   ExchangeToChain.AlmOKImmStopChain := TRUE;
   MecDetector.ScOk := FALSE;
   MecDetector.CycleOn := FALSE;
   MecDetector.Work := FALSE;
   MecDetector.OkToStop := FALSE;
   MecDetector.AlmOk := TRUE;
   MecDetector.MouldClear := FALSE;
   MecDetector.OutChainObstruction := FALSE;
   MecDetector.Ons_TimeWork := FALSE;
   MecDetector.SingleCycle := FALSE;
   MecDetector.Input.EnaSel := FALSE;
   MecDetector.Input.OffMouNotOpeSid := FALSE;
   MecDetector.Input.OnMouNotOpeSid := FALSE;
   MecDetector.Input.Chk1NotOpeSid := FALSE;
   MecDetector.Input.Chk2NotOpeSid := FALSE;
   MecDetector.Input.OffMouOpeSid := FALSE;
   MecDetector.Input.OnMouOpeSid := FALSE;
   MecDetector.Input.Chk1OpeSid := FALSE;
   MecDetector.Input.Chk2OpeSid := FALSE;
   MecDetector.Output.EnaSelLgh := FALSE;
   MecDetector.Output.CmdOnMouNotOpeSid := FALSE;
   MecDetector.Output.CmdOnMouOpeSid := FALSE;
   MecDetector.Man.Ons_SingleCycle := FALSE;
   MecDetector.Man.CmdSingleCycle := FALSE;
   MecDetector.Man.CmdOnMou := FALSE;
   MecDetector.Man.CmdOffMou := FALSE;
   MecDetector.Man.EnaPbt := FALSE;
   MecDetector.Man.RstCmd := FALSE;
   MecDetector.Man.ScreenNumber := 302_010_301;
   MecDetector.Man.WithinScreenRange := 0;
   MecDetector."Step"._00_CycleActivated_OnMouCmd := FALSE;
   MecDetector."Step"._10_OnMouPos_CheckResult := FALSE;
   MecDetector."Step"._20_ResultDone_OffMouCmd := FALSE;
   MecDetector."Step"._30_OffMouPos_EndCycle := FALSE;
   MecDetector."Step".Ons_StrobeWorkDone := FALSE;
   MecDetector."Step".StrobeWorkDone := FALSE;
   MecDetector."Step".ScSeqOk := FALSE;
   MecDetector."Step".SeqActive := FALSE;
   MecDetector."Step".TON_CheckResult.PT := T#500MS;
   MecDetector."Step".TON_CheckResult.IN := FALSE;
   MecDetector.RTO_Work.PT := T#1M;
   MecDetector.RTO_Work.IN := FALSE;
   MecDetector.TON_ScOK.PT := T#20S;
   MecDetector.TON_ScOK.IN := FALSE;
   MecDetector.TON_TimeoutWork.PT := T#20S;
   MecDetector.TON_TimeoutWork.IN := FALSE;
   MecDetector.TON_IncorrectPosOpeSide.PT := T#5S;
   MecDetector.TON_IncorrectPosOpeSide.IN := FALSE;
   MecDetector.TON_IncorrectPosNotOpeSide.PT := T#5S;
   MecDetector.TON_IncorrectPosNotOpeSide.IN := FALSE;
   MecDetector.TON_IncorrectPosPlate.PT := T#2S;
   MecDetector.TON_IncorrectPosPlate.IN := FALSE;
   OptDetector.ScOk := TRUE;
   OptDetector.CycleOn := FALSE;
   OptDetector.Work := FALSE;
   OptDetector.OkToStop := TRUE;
   OptDetector.AlmOk := TRUE;
   OptDetector.OutChainObstruction := TRUE;
   OptDetector.Ons_TimeWork := TRUE;
   OptDetector.Ons_ConnectionOn := FALSE;
   OptDetector.Ons_ChangeFormat := FALSE;
   OptDetector.Ons_RetrieveFormat := FALSE;
   OptDetector.RejectByDetector := FALSE;
   OptDetector.SingleCycle := FALSE;
   OptDetector.Ready := FALSE;
   OptDetector.SceneOk := FALSE;
   OptDetector.ChangeScene := FALSE;
   OptDetector.PhotoRequest := FALSE;
   OptDetector.SceneNumber := 0;
   OptDetector.Input.EnaSel := FALSE;
   OptDetector.Input.BrkSrs := TRUE;
   OptDetector.Input.Rdy := FALSE;
   OptDetector.Input.Brk := TRUE;
   OptDetector.Input.Run := TRUE;
   OptDetector.Input.Bsy := FALSE;
   OptDetector.Input.MouOk := FALSE;
   OptDetector.Input.Flt := FALSE;
   OptDetector.Input.WrkDone := FALSE;
   OptDetector.Input.FbkScn := 3;
   OptDetector.Output.EnaSelLgh := FALSE;
   OptDetector.Output.Lgh := FALSE;
   OptDetector.Output.CmdScnBit0 := TRUE;
   OptDetector.Output.CmdScnBit1 := FALSE;
   OptDetector.Output.CmdChgScn := FALSE;
   OptDetector.Output.CmdWrk := FALSE;
   OptDetector.Output.CmdRbo := FALSE;
   OptDetector.Output.CmdScn := 0;
   OptDetector.Man.Ons_SingleCycle := FALSE;
   OptDetector.Man.CmdSingleCycle := FALSE;
   OptDetector.Man.CmdStrobePhoto := FALSE;
   OptDetector.Man.EnaPbt := FALSE;
   OptDetector.Man.RstCmd := TRUE;
   OptDetector.Man.ScreenNumber := 302_020_301;
   OptDetector.Man.WithinScreenRange := 0;
   OptDetector."Step"._00_CycleActivated_StrobePhotoCmd := FALSE;
   OptDetector."Step"._10_ResultReady := FALSE;
   OptDetector."Step"._20_EndCycle := FALSE;
   OptDetector."Step".ons_StrobeWorkDone := FALSE;
   OptDetector."Step".StrobeWorkDone := FALSE;
   OptDetector."Step".ScSeqOk := FALSE;
   OptDetector."Step".SeqActive := FALSE;
   OptDetector.RTO_Work.PT := T#1M;
   OptDetector.RTO_Work.IN := FALSE;
   OptDetector.TON_ScOK.PT := T#20S;
   OptDetector.TON_ScOK.IN := FALSE;
   OptDetector.TON_TimeoutWork.PT := T#20S;
   OptDetector.TON_TimeoutWork.IN := FALSE;
   OptDetector.TON_TimeoutBusy.PT := T#5S;
   OptDetector.TON_TimeoutBusy.IN := FALSE;
   OptDetector.TON_TimeoutFormat.PT := T#5S;
   OptDetector.TON_TimeoutFormat.IN := FALSE;
   OptDetector.TOF_Ready.PT := T#500MS;
   OptDetector.TOF_Ready.ET := T#500MS;
   OptDetector.TOF_Ready.IN := FALSE;
   PusherExtractor.ScOk := FALSE;
   PusherExtractor.CycleOn := FALSE;
   PusherExtractor.Work := FALSE;
   PusherExtractor.OkToStop := FALSE;
   PusherExtractor.AlmOk := TRUE;
   PusherExtractor.DrivesEnabled := FALSE;
   PusherExtractor.OutChainObstruction := FALSE;
   PusherExtractor.SingleCycle := FALSE;
   PusherExtractor.RepositioningReq := FALSE;
   PusherExtractor.Ons_TimeWork := FALSE;
   PusherExtractor.NumMaxLevel := 0;
   PusherExtractor.Input.EnaSel := FALSE;
   PusherExtractor.Input.MaxLvl := FALSE;
   PusherExtractor.Input.HldOpnNotOpeSid := FALSE;
   PusherExtractor.Input.HldClsNotOpeSid := FALSE;
   PusherExtractor.Input.HldOpnOpeSid := FALSE;
   PusherExtractor.Input.HldClsOpeSid := FALSE;
   PusherExtractor.Output.EnaSelLgh := FALSE;
   PusherExtractor.Output.HldOpnNotOpeSid := FALSE;
   PusherExtractor.Output.HldClsNotOpeSid := FALSE;
   PusherExtractor.Output.HldOpnOpeSid := FALSE;
   PusherExtractor.Output.HldClsOpeSid := FALSE;
   PusherExtractor.Man.Ons_SingleCycle := FALSE;
   PusherExtractor.Man.CmdSupportOpen := FALSE;
   PusherExtractor.Man.CmdSupportClose := FALSE;
   PusherExtractor.Man.CmdSingleCycle := FALSE;
   PusherExtractor.Man.EnaPbt := FALSE;
   PusherExtractor.Man.RstCmd := FALSE;
   PusherExtractor.Man.ScreenNumber := 302_030_301;
   PusherExtractor.Man.WithinScreenRange := 0;
   PusherExtractor."Step"._00_CycleActived_UpCmd := FALSE;
   PusherExtractor."Step"._10_UpPos_IntermediateCmd := FALSE;
   PusherExtractor."Step"._20_IntermediatePos_OpenSupportCmd := FALSE;
   PusherExtractor."Step"._30_OpenSupportPos_DownCmd := FALSE;
   PusherExtractor."Step"._40_DownPos_CloseSupportCmd := FALSE;
   PusherExtractor."Step"._50_CloseSupportPos_CycleEnd := FALSE;
   PusherExtractor."Step".Ons_StrobeWorkDone := FALSE;
   PusherExtractor."Step".StrobeWorkDone := FALSE;
   PusherExtractor."Step".ScSeqOk := FALSE;
   PusherExtractor."Step".SeqActive := FALSE;
   PusherExtractor.Drive.AlmOk := FALSE;
   PusherExtractor.Drive.AlmEmerg := FALSE;
   PusherExtractor.Drive.AlmNode := FALSE;
   PusherExtractor.Drive.InitPosDrive := FALSE;
   PusherExtractor.Drive.InitPosDrivePLS := FALSE;
   PusherExtractor.Drive.GearingON := FALSE;
   PusherExtractor.Drive.CamHook := FALSE;
   PusherExtractor.Drive.CamStoppingPhase := FALSE;
   PusherExtractor.Drive.RepositioningRequest := FALSE;
   PusherExtractor.Drive.CamRequestResult := FALSE;
   PusherExtractor.Drive.CamRequestError := FALSE;
   PusherExtractor.Drive.CamRequestOk := FALSE;
   PusherExtractor.Drive.CalibDisAxisReq := FALSE;
   PusherExtractor.Drive.CalibReq := FALSE;
   PusherExtractor.Drive.CalibProcess := FALSE;
   PusherExtractor.Drive.HwOvertravelDisReq := FALSE;
   PusherExtractor.Drive.HwOvertravelEnReq := FALSE;
   PusherExtractor.Drive.AuxCamRequest := FALSE;
   PusherExtractor.Drive.TorquePeakEna := FALSE;
   PusherExtractor.Drive.Cmd_Repos := FALSE;
   PusherExtractor.Drive.Ons_CamRequest := FALSE;
   PusherExtractor.Drive.AuxCmdPosition := 0;
   PusherExtractor.Drive.Unwind := 0.0;
   PusherExtractor.Drive.MaxDev := 0.0;
   PusherExtractor.Drive.ReposSpeed := 100.0;
   PusherExtractor.Drive.CalcSlaveDifferenceABS := 0.0;
   PusherExtractor.Drive.CalcModPosition := 0.0;
   PusherExtractor.Drive.CalcSlaveDifference := 0.0;
   PusherExtractor.Drive.CalcMinDeltaPos := 0.0;
   PusherExtractor.Drive.CalcMaxDeltaPos := 0.0;
   PusherExtractor.Drive.CalcHalfPosUnwind := 0.0;
   PusherExtractor.Drive.Man.Cmd_PosJog := FALSE;
   PusherExtractor.Drive.Man.Cmd_NegJog := FALSE;
   PusherExtractor.Drive.Man.Cmd_Step := FALSE;
   PusherExtractor.Drive.Man.Cmd_Forward := FALSE;
   PusherExtractor.Drive.Man.Cmd_Backward := FALSE;
   PusherExtractor.Drive.Man.Cmd_Up := FALSE;
   PusherExtractor.Drive.Man.Cmd_Down := FALSE;
   PusherExtractor.Drive.Man.Cmd_Intermediate := FALSE;
   PusherExtractor.Drive.Man.Cmd_Open := FALSE;
   PusherExtractor.Drive.Man.Cmd_Close := FALSE;
   PusherExtractor.Drive.Man.Cmd_PreOpen := FALSE;
   PusherExtractor.Drive.Man.Cmd_Maintenance := FALSE;
   PusherExtractor.Drive.Man.Cmd_OperatorSide := FALSE;
   PusherExtractor.Drive.Man.Cmd_NotOperatorSide := FALSE;
   PusherExtractor.Drive.Man.Cmd_OnMould := FALSE;
   PusherExtractor.Drive.Man.Cmd_OffMould := FALSE;
   PusherExtractor.Drive.Man.Cmd_Pos0 := FALSE;
   PusherExtractor.Drive.Man.Cmd_Pos1 := FALSE;
   PusherExtractor.Drive.Man.Cmd_Pos2 := FALSE;
   PusherExtractor.Drive.Man.Cmd_Pos3 := FALSE;
   PusherExtractor.Drive.Man.Cmd_Pos4 := FALSE;
   PusherExtractor.Drive.Man.Cmd_Pos5 := FALSE;
   PusherExtractor.Drive.Man.Ons_Step := FALSE;
   PusherExtractor.Drive.Man.PhaseJogCmd := FALSE;
   PusherExtractor.Drive.Man.CmdStartStep := FALSE;
   PusherExtractor.Drive.Man.CmdEndStep := FALSE;
   PusherExtractor.Drive.Man.StepCond := FALSE;
   PusherExtractor.Drive.Man.TON_DelayHomeCmd.PT := T#3S;
   PusherExtractor.Drive.Man.TON_DelayHomeCmd.IN := FALSE;
   PusherExtractor.Drive.Auto.Cmd_Step := FALSE;
   PusherExtractor.Drive.Auto.Cmd_StartStep := FALSE;
   PusherExtractor.Drive.Auto.Cmd_EndStep := FALSE;
   PusherExtractor.Drive.Auto.Cmd_Forward := FALSE;
   PusherExtractor.Drive.Auto.Cmd_Backward := FALSE;
   PusherExtractor.Drive.Auto.Cmd_Up := FALSE;
   PusherExtractor.Drive.Auto.Cmd_Down := FALSE;
   PusherExtractor.Drive.Auto.Cmd_Intermediate := FALSE;
   PusherExtractor.Drive.Auto.Cmd_Open := FALSE;
   PusherExtractor.Drive.Auto.Cmd_Close := FALSE;
   PusherExtractor.Drive.Auto.Cmd_PreOpen := FALSE;
   PusherExtractor.Drive.Auto.Cmd_Maintenance := FALSE;
   PusherExtractor.Drive.Auto.Cmd_OperatorSide := FALSE;
   PusherExtractor.Drive.Auto.Cmd_NotOperatorSide := FALSE;
   PusherExtractor.Drive.Auto.Cmd_OnMould := FALSE;
   PusherExtractor.Drive.Auto.Cmd_OffMould := FALSE;
   PusherExtractor.Drive.Auto.Cmd_Pos0 := FALSE;
   PusherExtractor.Drive.Auto.Cmd_Pos1 := FALSE;
   PusherExtractor.Drive.Auto.Cmd_Pos2 := FALSE;
   PusherExtractor.Drive.Auto.Cmd_Pos3 := FALSE;
   PusherExtractor.Drive.Auto.Cmd_Pos4 := FALSE;
   PusherExtractor.Drive.Auto.Cmd_Pos5 := FALSE;
   PusherExtractor.Drive.Auto.Cmd_Gear := FALSE;
   PusherExtractor.Drive.ACT.CMD.Enable := FALSE;
   PusherExtractor.Drive.ACT.CMD.Pos_Mode := FALSE;
   PusherExtractor.Drive.ACT.CMD.MergeDisabled := FALSE;
   PusherExtractor.Drive.ACT.CMD.SCurve := FALSE;
   PusherExtractor.Drive.ACT.CMD.Cam_Mode := FALSE;
   PusherExtractor.Drive.ACT.CMD.Cam_Request := FALSE;
   PusherExtractor.Drive.ACT.CMD.Cam_PhaseStop := FALSE;
   PusherExtractor.Drive.ACT.CMD.Gear_Mode := FALSE;
   PusherExtractor.Drive.ACT.CMD.Repos_Req := FALSE;
   PusherExtractor.Drive.ACT.CMD.Jog_Pos := FALSE;
   PusherExtractor.Drive.ACT.CMD.Jog_Neg := FALSE;
   PusherExtractor.Drive.ACT.CMD.Stop := FALSE;
   PusherExtractor.Drive.ACT.CMD.Calibration_Req := FALSE;
   PusherExtractor.Drive.ACT.CMD.Reset := FALSE;
   PusherExtractor.Drive.ACT.CMD.RegInput1 := FALSE;
   PusherExtractor.Drive.ACT.CMD.Brake_Release := FALSE;
   PusherExtractor.Drive.ACT.CMD.HwPosOvertravel_Dis := FALSE;
   PusherExtractor.Drive.ACT.CMD.HwNegOvertravel_Dis := FALSE;
   PusherExtractor.Drive.ACT.CMD.HwOvertravel_MSG_En := FALSE;
   PusherExtractor.Drive.ACT.CMD.OneShootMove := FALSE;
   PusherExtractor.Drive.ACT.CMD.Move_Type := 0;
   PusherExtractor.Drive.ACT.CMD.Target_Pos := 0.0;
   PusherExtractor.Drive.ACT.CMD.Speed := 0.0;
   PusherExtractor.Drive.ACT.CMD.Acceleration := 0.0;
   PusherExtractor.Drive.ACT.CMD.Deceleration := 0.0;
   PusherExtractor.Drive.ACT.CMD.Torque_Limit := 0.0;
   PusherExtractor.Drive.ACT.CMD.Gear_Ratio := 0.0;
   PusherExtractor.Drive.ACT.CMD.Mccp_Length := 0;
   PusherExtractor.Drive.ACT.CMD.Mccp_StartSlope := 0.0;
   PusherExtractor.Drive.ACT.CMD.Mccp_EndSlope := 0.0;
   PusherExtractor.Drive.ACT.CMD.Mapc_Direction := 0;
   PusherExtractor.Drive.ACT.CMD.Mapc_SlaveScaling := 0.0;
   PusherExtractor.Drive.ACT.CMD.Mapc_MasterScaling := 0.0;
   PusherExtractor.Drive.ACT.CMD.Mapc_MasterLockPosition := 0.0;
   PusherExtractor.Drive.ACT.CMD.Mapc_CamLockPosition := 0.0;
   PusherExtractor.Drive.ACT.CMD.Cam[0..39].leadingValueStart := 0.0;
   PusherExtractor.Drive.ACT.CMD.Cam[0..39].leadingValueEnd := 0.0;
   PusherExtractor.Drive.ACT.CMD.Cam[0..39].followingValueStart := 0.0;
   PusherExtractor.Drive.ACT.CMD.Cam[0..39].followingValueEnd := 0.0;
   PusherExtractor.Drive.ACT.CMD.Cam[0..39].geoVeloStart := 0.0;
   PusherExtractor.Drive.ACT.CMD.Cam[0..39].geoVeloEnd := 0.0;
   PusherExtractor.Drive.ACT.CMD.Cam[0..39].geoAccelStart := 0.0;
   PusherExtractor.Drive.ACT.CMD.Cam[0..39].geoAccelEnd := 0.0;
   PusherExtractor.Drive.ACT.CMD.Cam[0..39].geoJerkStart := 0.0;
   PusherExtractor.Drive.ACT.CMD.Cam[0..39].geoJerkEnd := 0.0;
   PusherExtractor.Drive.ACT.CMD.Cam[0..39].inflectionPointParameter := 0.5;
   PusherExtractor.Drive.ACT.CMD.Cam[0..39].modVeloTrapezoidParameter := 1.0;
   PusherExtractor.Drive.ACT.CMD.Cam[0..39].modSineMaxAccelCaStar := 0.0;
   PusherExtractor.Drive.ACT.CMD.Cam[0..39].camProfileType := 0;
   PusherExtractor.Drive.ACT.FBK.Ready := FALSE;
   PusherExtractor.Drive.ACT.FBK.Calibrated := FALSE;
   PusherExtractor.Drive.ACT.FBK.Fault := FALSE;
   PusherExtractor.Drive.ACT.FBK.ModuleConnFault := FALSE;
   PusherExtractor.Drive.ACT.FBK.In_Position := FALSE;
   PusherExtractor.Drive.ACT.FBK.Standstill := FALSE;
   PusherExtractor.Drive.ACT.FBK.Enabled := FALSE;
   PusherExtractor.Drive.ACT.FBK.BusReadyStatus := FALSE;
   PusherExtractor.Drive.ACT.FBK.BrakeReleased := FALSE;
   PusherExtractor.Drive.ACT.FBK.HwPosOvertravelDisabled := FALSE;
   PusherExtractor.Drive.ACT.FBK.HwNegOvertravelDisabled := FALSE;
   PusherExtractor.Drive.ACT.FBK.SafeOffStatus := FALSE;
   PusherExtractor.Drive.ACT.FBK.MaxTorqueLimit := FALSE;
   PusherExtractor.Drive.ACT.FBK.PosMerge_IP := FALSE;
   PusherExtractor.Drive.ACT.FBK.PosMerge_PC := FALSE;
   PusherExtractor.Drive.ACT.FBK.Gearing_IP := FALSE;
   PusherExtractor.Drive.ACT.FBK.Position := 0.0;
   PusherExtractor.Drive.ACT.FBK.Speed := 0.0;
   PusherExtractor.Drive.ACT.FBK.Torque := 0.0;
   PusherExtractor.Drive.ACT.FBK.RegInput1Pos := 0.0;
   PusherExtractor.Drive.ACT.FBK.SeqCamErrorCode := 0;
   PusherExtractor.Drive.ACT.FBK.SeqCamTargetPosMAM := 0.0;
   PusherExtractor.Drive.ACT.FBK.SeqCamStatus.EndSequence := FALSE;
   PusherExtractor.Drive.ACT.FBK.SeqCamStatus.EndSuccess := FALSE;
   PusherExtractor.Drive.ACT.FBK.SeqCamStatus.EndError := FALSE;
   PusherExtractor.Drive.ACT.FBK.SeqCamStatus.CamHook := FALSE;
   PusherExtractor.Drive.ACT.FBK.SeqCamStatus.BothMapc_IP := FALSE;
   PusherExtractor.Drive.ACT.FBK.SeqCamStatus.SlaveFwd := FALSE;
   PusherExtractor.Drive.ACT.FBK.SeqCamStatus.SlaveBwd := FALSE;
   PusherExtractor.Drive.ACT.FBK.SeqCamStatus.SlaveUnwind := FALSE;
   PusherExtractor.Drive.ACT.FBK.SeqCamStatus.WaitValidByOpe := FALSE;
   PusherExtractor.Drive.ACT.FBK.SeqCamStatus.MapcA_IP := FALSE;
   PusherExtractor.Drive.ACT.FBK.SeqCamStatus.MapcB_IP := FALSE;
   PusherExtractor.Drive.ACT.FBK.SeqCamStatus.MapcC_IP := FALSE;
   PusherExtractor.Drive.ACT.FBK.SeqCamStatus.CamOnce_PC := FALSE;
   PusherExtractor.Drive.ACT.FBK.SeqCamStatus.MaxDevError := FALSE;
   PusherExtractor.Drive.ACT.FBK.SeqCamStatus.PositionCamLockStatus := FALSE;
   PusherExtractor.Drive.ACT.FBK.SeqCamStatus.WaitRestart := FALSE;
   PusherExtractor.Drive.ACT.FBK.SeqCamStatus.Bit17 := FALSE;
   PusherExtractor.Drive.ACT.FBK.SeqCamStatus.Bit18 := FALSE;
   PusherExtractor.Drive.ACT.FBK.SeqCamStatus.Bit19 := FALSE;
   PusherExtractor.Drive.ACT.FBK.SeqCamStatus.Bit20 := FALSE;
   PusherExtractor.Drive.ACT.FBK.SeqCamStatus.Bit21 := FALSE;
   PusherExtractor.Drive.ACT.FBK.SeqCamStatus.Bit22 := FALSE;
   PusherExtractor.Drive.ACT.FBK.SeqCamStatus.Bit23 := FALSE;
   PusherExtractor.Drive.ACT.FBK.SeqCamStatus.Bit24 := FALSE;
   PusherExtractor.Drive.ACT.FBK.SeqCamStatus.Bit25 := FALSE;
   PusherExtractor.Drive.ACT.FBK.SeqCamStatus.Bit26 := FALSE;
   PusherExtractor.Drive.ACT.FBK.SeqCamStatus.Bit27 := FALSE;
   PusherExtractor.Drive.ACT.FBK.SeqCamStatus.Bit28 := FALSE;
   PusherExtractor.Drive.ACT.FBK.SeqCamStatus.Bit29 := FALSE;
   PusherExtractor.Drive.ACT.FBK.SeqCamStatus.Bit30 := FALSE;
   PusherExtractor.Drive.ACT.FBK.SeqCamStatus.Bit31 := FALSE;
   PusherExtractor.Drive.ACT.FBK.SeqCamStatus.Bit32 := FALSE;
   PusherExtractor.Drive.PLS.FinePosOk.LowLimit := 0.0;
   PusherExtractor.Drive.PLS.FinePosOk.HighLimit := 0.0;
   PusherExtractor.Drive.PLS.FinePosOk.Ok := FALSE;
   PusherExtractor.Drive.PLS.KeepPosOk.LowLimit := 0.0;
   PusherExtractor.Drive.PLS.KeepPosOk.HighLimit := 0.0;
   PusherExtractor.Drive.PLS.KeepPosOk.Ok := FALSE;
   PusherExtractor.Drive.PLS.Up.LowLimit := 0.0;
   PusherExtractor.Drive.PLS.Up.HighLimit := 0.0;
   PusherExtractor.Drive.PLS.Up.Ok := FALSE;
   PusherExtractor.Drive.PLS.Intermediate.LowLimit := 0.0;
   PusherExtractor.Drive.PLS.Intermediate.HighLimit := 0.0;
   PusherExtractor.Drive.PLS.Intermediate.Ok := FALSE;
   PusherExtractor.Drive.PLS.Down.LowLimit := 0.0;
   PusherExtractor.Drive.PLS.Down.HighLimit := 0.0;
   PusherExtractor.Drive.PLS.Down.Ok := FALSE;
   PusherExtractor.Drive.PLS.Forward.LowLimit := 0.0;
   PusherExtractor.Drive.PLS.Forward.HighLimit := 0.0;
   PusherExtractor.Drive.PLS.Forward.Ok := FALSE;
   PusherExtractor.Drive.PLS.Backward.LowLimit := 0.0;
   PusherExtractor.Drive.PLS.Backward.HighLimit := 0.0;
   PusherExtractor.Drive.PLS.Backward.Ok := FALSE;
   PusherExtractor.Drive.PLS.Open.LowLimit := 0.0;
   PusherExtractor.Drive.PLS.Open.HighLimit := 0.0;
   PusherExtractor.Drive.PLS.Open.Ok := FALSE;
   PusherExtractor.Drive.PLS.Close.LowLimit := 0.0;
   PusherExtractor.Drive.PLS.Close.HighLimit := 0.0;
   PusherExtractor.Drive.PLS.Close.Ok := FALSE;
   PusherExtractor.Drive.PLS.PreOpen.LowLimit := 0.0;
   PusherExtractor.Drive.PLS.PreOpen.HighLimit := 0.0;
   PusherExtractor.Drive.PLS.PreOpen.Ok := FALSE;
   PusherExtractor.Drive.PLS.Maintenance.LowLimit := 0.0;
   PusherExtractor.Drive.PLS.Maintenance.HighLimit := 0.0;
   PusherExtractor.Drive.PLS.Maintenance.Ok := FALSE;
   PusherExtractor.Drive.PLS.OperatorSide.LowLimit := 0.0;
   PusherExtractor.Drive.PLS.OperatorSide.HighLimit := 0.0;
   PusherExtractor.Drive.PLS.OperatorSide.Ok := FALSE;
   PusherExtractor.Drive.PLS.NotOperatorSide.LowLimit := 0.0;
   PusherExtractor.Drive.PLS.NotOperatorSide.HighLimit := 0.0;
   PusherExtractor.Drive.PLS.NotOperatorSide.Ok := FALSE;
   PusherExtractor.Drive.PLS.OnMould.LowLimit := 0.0;
   PusherExtractor.Drive.PLS.OnMould.HighLimit := 0.0;
   PusherExtractor.Drive.PLS.OnMould.Ok := FALSE;
   PusherExtractor.Drive.PLS.OffMould.LowLimit := 0.0;
   PusherExtractor.Drive.PLS.OffMould.HighLimit := 0.0;
   PusherExtractor.Drive.PLS.OffMould.Ok := FALSE;
   PusherExtractor.Drive.PLS.Pos0.LowLimit := 0.0;
   PusherExtractor.Drive.PLS.Pos0.HighLimit := 0.0;
   PusherExtractor.Drive.PLS.Pos0.Ok := FALSE;
   PusherExtractor.Drive.PLS.Pos1.LowLimit := 0.0;
   PusherExtractor.Drive.PLS.Pos1.HighLimit := 0.0;
   PusherExtractor.Drive.PLS.Pos1.Ok := FALSE;
   PusherExtractor.Drive.PLS.Pos2.LowLimit := 0.0;
   PusherExtractor.Drive.PLS.Pos2.HighLimit := 0.0;
   PusherExtractor.Drive.PLS.Pos2.Ok := FALSE;
   PusherExtractor.Drive.PLS.Pos3.LowLimit := 0.0;
   PusherExtractor.Drive.PLS.Pos3.HighLimit := 0.0;
   PusherExtractor.Drive.PLS.Pos3.Ok := FALSE;
   PusherExtractor.Drive.PLS.Pos4.LowLimit := 0.0;
   PusherExtractor.Drive.PLS.Pos4.HighLimit := 0.0;
   PusherExtractor.Drive.PLS.Pos4.Ok := FALSE;
   PusherExtractor.Drive.PLS.Pos5.LowLimit := 0.0;
   PusherExtractor.Drive.PLS.Pos5.HighLimit := 0.0;
   PusherExtractor.Drive.PLS.Pos5.Ok := FALSE;
   PusherExtractor.Drive.TON_EnableDrive.PT := T#500MS;
   PusherExtractor.Drive.TON_EnableDrive.IN := FALSE;
   PusherExtractor.Drive.TON_HwOvertravel_Dis.PT := T#0MS;
   PusherExtractor.Drive.TON_HwOvertravel_Dis.IN := FALSE;
   PusherExtractor.Drive.TON_HwOvertravel_En.PT := T#0MS;
   PusherExtractor.Drive.TON_HwOvertravel_En.IN := FALSE;
   PusherExtractor.Drive.TON_TimeoutMovement.PT := T#8S;
   PusherExtractor.Drive.TON_TimeoutMovement.IN := FALSE;
   PusherExtractor.TON_ResetMaxLevel.PT := T#2S;
   PusherExtractor.TON_ResetMaxLevel.IN := FALSE;
   PusherExtractor.RTO_Work.PT := T#1M;
   PusherExtractor.RTO_Work.IN := FALSE;
   PusherExtractor.TON_ScOK.PT := T#20S;
   PusherExtractor.TON_ScOK.IN := FALSE;
   PusherExtractor.TON_IncorrectPosOpeSide.PT := T#4S;
   PusherExtractor.TON_IncorrectPosOpeSide.IN := FALSE;
   PusherExtractor.TON_IncorrectPosNotOpeSide.PT := T#4S;
   PusherExtractor.TON_IncorrectPosNotOpeSide.IN := FALSE;
   PusherExtractor.TON_Sign_MaxLevel.PT := T#1S;
   PusherExtractor.TON_Sign_MaxLevel.IN := FALSE;
   PusherExtractor.TON_TimeoutWork.PT := T#20S;
   PusherExtractor.TON_TimeoutWork.IN := FALSE;
   RotaryExtractor.ScOk := FALSE;
   RotaryExtractor.CycleOn := FALSE;
   RotaryExtractor.Work := FALSE;
   RotaryExtractor.OkToStop := TRUE;
   RotaryExtractor.AlmOk := TRUE;
   RotaryExtractor.DrivesEnabled := FALSE;
   RotaryExtractor.OutChainObstruction := TRUE;
   RotaryExtractor.RepositioningReq := FALSE;
   RotaryExtractor.Ons_TimeWork := TRUE;
   RotaryExtractor.NumMaxLevel := 0;
   RotaryExtractor.Input.EnaSel := FALSE;
   RotaryExtractor.Input.MaxLvl := FALSE;
   RotaryExtractor.Output.EnaSelLgh := FALSE;
   RotaryExtractor.Man.EnaPbt := FALSE;
   RotaryExtractor.Man.RstCmd := TRUE;
   RotaryExtractor.Man.ScreenNumber := 302_040_301;
   RotaryExtractor.Man.WithinScreenRange := 0;
   RotaryExtractor."Step"._00_CycleActived_StartRotationCmd := FALSE;
   RotaryExtractor."Step"._10_RotationOutPos_StopRotationCmd := FALSE;
   RotaryExtractor."Step"._20_FinePos_CycleEnd := FALSE;
   RotaryExtractor."Step".Ons_StrobeWorkDone := FALSE;
   RotaryExtractor."Step".StrobeWorkDone := FALSE;
   RotaryExtractor."Step".ScSeqOk := FALSE;
   RotaryExtractor."Step".SeqActive := FALSE;
   RotaryExtractor.Drive.AlmOk := FALSE;
   RotaryExtractor.Drive.AlmEmerg := FALSE;
   RotaryExtractor.Drive.AlmNode := FALSE;
   RotaryExtractor.Drive.InitPosDrive := FALSE;
   RotaryExtractor.Drive.InitPosDrivePLS := FALSE;
   RotaryExtractor.Drive.GearingON := FALSE;
   RotaryExtractor.Drive.CamHook := FALSE;
   RotaryExtractor.Drive.CamStoppingPhase := FALSE;
   RotaryExtractor.Drive.RepositioningRequest := FALSE;
   RotaryExtractor.Drive.CamRequestResult := FALSE;
   RotaryExtractor.Drive.CamRequestError := FALSE;
   RotaryExtractor.Drive.CamRequestOk := FALSE;
   RotaryExtractor.Drive.CalibDisAxisReq := FALSE;
   RotaryExtractor.Drive.CalibReq := FALSE;
   RotaryExtractor.Drive.CalibProcess := FALSE;
   RotaryExtractor.Drive.HwOvertravelDisReq := FALSE;
   RotaryExtractor.Drive.HwOvertravelEnReq := FALSE;
   RotaryExtractor.Drive.AuxCamRequest := FALSE;
   RotaryExtractor.Drive.TorquePeakEna := TRUE;
   RotaryExtractor.Drive.Cmd_Repos := FALSE;
   RotaryExtractor.Drive.Ons_CamRequest := FALSE;
   RotaryExtractor.Drive.AuxCmdPosition := 0;
   RotaryExtractor.Drive.Unwind := 120.0;
   RotaryExtractor.Drive.MaxDev := 0.0;
   RotaryExtractor.Drive.ReposSpeed := 100.0;
   RotaryExtractor.Drive.CalcSlaveDifferenceABS := 0.0;
   RotaryExtractor.Drive.CalcModPosition := 0.0;
   RotaryExtractor.Drive.CalcSlaveDifference := 0.0;
   RotaryExtractor.Drive.CalcMinDeltaPos := 0.0;
   RotaryExtractor.Drive.CalcMaxDeltaPos := 0.0;
   RotaryExtractor.Drive.CalcHalfPosUnwind := 0.0;
   RotaryExtractor.Drive.Man.Cmd_PosJog := FALSE;
   RotaryExtractor.Drive.Man.Cmd_NegJog := FALSE;
   RotaryExtractor.Drive.Man.Cmd_Step := FALSE;
   RotaryExtractor.Drive.Man.Cmd_Forward := FALSE;
   RotaryExtractor.Drive.Man.Cmd_Backward := FALSE;
   RotaryExtractor.Drive.Man.Cmd_Up := FALSE;
   RotaryExtractor.Drive.Man.Cmd_Down := FALSE;
   RotaryExtractor.Drive.Man.Cmd_Intermediate := FALSE;
   RotaryExtractor.Drive.Man.Cmd_Open := FALSE;
   RotaryExtractor.Drive.Man.Cmd_Close := FALSE;
   RotaryExtractor.Drive.Man.Cmd_PreOpen := FALSE;
   RotaryExtractor.Drive.Man.Cmd_Maintenance := FALSE;
   RotaryExtractor.Drive.Man.Cmd_OperatorSide := FALSE;
   RotaryExtractor.Drive.Man.Cmd_NotOperatorSide := FALSE;
   RotaryExtractor.Drive.Man.Cmd_OnMould := FALSE;
   RotaryExtractor.Drive.Man.Cmd_OffMould := FALSE;
   RotaryExtractor.Drive.Man.Cmd_Pos0 := FALSE;
   RotaryExtractor.Drive.Man.Cmd_Pos1 := FALSE;
   RotaryExtractor.Drive.Man.Cmd_Pos2 := FALSE;
   RotaryExtractor.Drive.Man.Cmd_Pos3 := FALSE;
   RotaryExtractor.Drive.Man.Cmd_Pos4 := FALSE;
   RotaryExtractor.Drive.Man.Cmd_Pos5 := FALSE;
   RotaryExtractor.Drive.Man.Ons_Step := FALSE;
   RotaryExtractor.Drive.Man.PhaseJogCmd := FALSE;
   RotaryExtractor.Drive.Man.CmdStartStep := FALSE;
   RotaryExtractor.Drive.Man.CmdEndStep := FALSE;
   RotaryExtractor.Drive.Man.StepCond := FALSE;
   RotaryExtractor.Drive.Man.TON_DelayHomeCmd.PT := T#3S;
   RotaryExtractor.Drive.Man.TON_DelayHomeCmd.IN := FALSE;
   RotaryExtractor.Drive.Auto.Cmd_Step := FALSE;
   RotaryExtractor.Drive.Auto.Cmd_StartStep := FALSE;
   RotaryExtractor.Drive.Auto.Cmd_EndStep := FALSE;
   RotaryExtractor.Drive.Auto.Cmd_Forward := FALSE;
   RotaryExtractor.Drive.Auto.Cmd_Backward := FALSE;
   RotaryExtractor.Drive.Auto.Cmd_Up := FALSE;
   RotaryExtractor.Drive.Auto.Cmd_Down := FALSE;
   RotaryExtractor.Drive.Auto.Cmd_Intermediate := FALSE;
   RotaryExtractor.Drive.Auto.Cmd_Open := FALSE;
   RotaryExtractor.Drive.Auto.Cmd_Close := FALSE;
   RotaryExtractor.Drive.Auto.Cmd_PreOpen := FALSE;
   RotaryExtractor.Drive.Auto.Cmd_Maintenance := FALSE;
   RotaryExtractor.Drive.Auto.Cmd_OperatorSide := FALSE;
   RotaryExtractor.Drive.Auto.Cmd_NotOperatorSide := FALSE;
   RotaryExtractor.Drive.Auto.Cmd_OnMould := FALSE;
   RotaryExtractor.Drive.Auto.Cmd_OffMould := FALSE;
   RotaryExtractor.Drive.Auto.Cmd_Pos0 := FALSE;
   RotaryExtractor.Drive.Auto.Cmd_Pos1 := FALSE;
   RotaryExtractor.Drive.Auto.Cmd_Pos2 := FALSE;
   RotaryExtractor.Drive.Auto.Cmd_Pos3 := FALSE;
   RotaryExtractor.Drive.Auto.Cmd_Pos4 := FALSE;
   RotaryExtractor.Drive.Auto.Cmd_Pos5 := FALSE;
   RotaryExtractor.Drive.Auto.Cmd_Gear := FALSE;
   RotaryExtractor.Drive.ACT.CMD.Enable := FALSE;
   RotaryExtractor.Drive.ACT.CMD.Pos_Mode := FALSE;
   RotaryExtractor.Drive.ACT.CMD.MergeDisabled := FALSE;
   RotaryExtractor.Drive.ACT.CMD.SCurve := FALSE;
   RotaryExtractor.Drive.ACT.CMD.Cam_Mode := FALSE;
   RotaryExtractor.Drive.ACT.CMD.Cam_Request := FALSE;
   RotaryExtractor.Drive.ACT.CMD.Cam_PhaseStop := FALSE;
   RotaryExtractor.Drive.ACT.CMD.Gear_Mode := FALSE;
   RotaryExtractor.Drive.ACT.CMD.Repos_Req := FALSE;
   RotaryExtractor.Drive.ACT.CMD.Jog_Pos := FALSE;
   RotaryExtractor.Drive.ACT.CMD.Jog_Neg := FALSE;
   RotaryExtractor.Drive.ACT.CMD.Stop := TRUE;
   RotaryExtractor.Drive.ACT.CMD.Calibration_Req := FALSE;
   RotaryExtractor.Drive.ACT.CMD.Reset := FALSE;
   RotaryExtractor.Drive.ACT.CMD.RegInput1 := FALSE;
   RotaryExtractor.Drive.ACT.CMD.Brake_Release := FALSE;
   RotaryExtractor.Drive.ACT.CMD.HwPosOvertravel_Dis := FALSE;
   RotaryExtractor.Drive.ACT.CMD.HwNegOvertravel_Dis := FALSE;
   RotaryExtractor.Drive.ACT.CMD.HwOvertravel_MSG_En := FALSE;
   RotaryExtractor.Drive.ACT.CMD.OneShootMove := FALSE;
   RotaryExtractor.Drive.ACT.CMD.Move_Type := 0;
   RotaryExtractor.Drive.ACT.CMD.Target_Pos := 0.0;
   RotaryExtractor.Drive.ACT.CMD.Speed := 0.0;
   RotaryExtractor.Drive.ACT.CMD.Acceleration := 0.0;
   RotaryExtractor.Drive.ACT.CMD.Deceleration := 4500.0;
   RotaryExtractor.Drive.ACT.CMD.Torque_Limit := 30.0;
   RotaryExtractor.Drive.ACT.CMD.Gear_Ratio := 0.0;
   RotaryExtractor.Drive.ACT.CMD.Mccp_Length := 0;
   RotaryExtractor.Drive.ACT.CMD.Mccp_StartSlope := 0.0;
   RotaryExtractor.Drive.ACT.CMD.Mccp_EndSlope := 0.0;
   RotaryExtractor.Drive.ACT.CMD.Mapc_Direction := 0;
   RotaryExtractor.Drive.ACT.CMD.Mapc_SlaveScaling := 0.0;
   RotaryExtractor.Drive.ACT.CMD.Mapc_MasterScaling := 0.0;
   RotaryExtractor.Drive.ACT.CMD.Mapc_MasterLockPosition := 0.0;
   RotaryExtractor.Drive.ACT.CMD.Mapc_CamLockPosition := 0.0;
   RotaryExtractor.Drive.ACT.CMD.Cam[0..39].leadingValueStart := 0.0;
   RotaryExtractor.Drive.ACT.CMD.Cam[0..39].leadingValueEnd := 0.0;
   RotaryExtractor.Drive.ACT.CMD.Cam[0..39].followingValueStart := 0.0;
   RotaryExtractor.Drive.ACT.CMD.Cam[0..39].followingValueEnd := 0.0;
   RotaryExtractor.Drive.ACT.CMD.Cam[0..39].geoVeloStart := 0.0;
   RotaryExtractor.Drive.ACT.CMD.Cam[0..39].geoVeloEnd := 0.0;
   RotaryExtractor.Drive.ACT.CMD.Cam[0..39].geoAccelStart := 0.0;
   RotaryExtractor.Drive.ACT.CMD.Cam[0..39].geoAccelEnd := 0.0;
   RotaryExtractor.Drive.ACT.CMD.Cam[0..39].geoJerkStart := 0.0;
   RotaryExtractor.Drive.ACT.CMD.Cam[0..39].geoJerkEnd := 0.0;
   RotaryExtractor.Drive.ACT.CMD.Cam[0..39].inflectionPointParameter := 0.5;
   RotaryExtractor.Drive.ACT.CMD.Cam[0..39].modVeloTrapezoidParameter := 1.0;
   RotaryExtractor.Drive.ACT.CMD.Cam[0..39].modSineMaxAccelCaStar := 0.0;
   RotaryExtractor.Drive.ACT.CMD.Cam[0..39].camProfileType := 0;
   RotaryExtractor.Drive.ACT.FBK.Ready := TRUE;
   RotaryExtractor.Drive.ACT.FBK.Calibrated := TRUE;
   RotaryExtractor.Drive.ACT.FBK.Fault := FALSE;
   RotaryExtractor.Drive.ACT.FBK.ModuleConnFault := FALSE;
   RotaryExtractor.Drive.ACT.FBK.In_Position := FALSE;
   RotaryExtractor.Drive.ACT.FBK.Standstill := TRUE;
   RotaryExtractor.Drive.ACT.FBK.Enabled := FALSE;
   RotaryExtractor.Drive.ACT.FBK.BusReadyStatus := FALSE;
   RotaryExtractor.Drive.ACT.FBK.BrakeReleased := FALSE;
   RotaryExtractor.Drive.ACT.FBK.HwPosOvertravelDisabled := FALSE;
   RotaryExtractor.Drive.ACT.FBK.HwNegOvertravelDisabled := FALSE;
   RotaryExtractor.Drive.ACT.FBK.SafeOffStatus := FALSE;
   RotaryExtractor.Drive.ACT.FBK.MaxTorqueLimit := FALSE;
   RotaryExtractor.Drive.ACT.FBK.PosMerge_IP := FALSE;
   RotaryExtractor.Drive.ACT.FBK.PosMerge_PC := FALSE;
   RotaryExtractor.Drive.ACT.FBK.Gearing_IP := FALSE;
   RotaryExtractor.Drive.ACT.FBK.Position := 0.003;
   RotaryExtractor.Drive.ACT.FBK.Speed := 0.0;
   RotaryExtractor.Drive.ACT.FBK.Torque := 0.0;
   RotaryExtractor.Drive.ACT.FBK.RegInput1Pos := 0.0;
   RotaryExtractor.Drive.ACT.FBK.SeqCamErrorCode := 0;
   RotaryExtractor.Drive.ACT.FBK.SeqCamTargetPosMAM := 0.0;
   RotaryExtractor.Drive.ACT.FBK.SeqCamStatus.EndSequence := FALSE;
   RotaryExtractor.Drive.ACT.FBK.SeqCamStatus.EndSuccess := FALSE;
   RotaryExtractor.Drive.ACT.FBK.SeqCamStatus.EndError := FALSE;
   RotaryExtractor.Drive.ACT.FBK.SeqCamStatus.CamHook := FALSE;
   RotaryExtractor.Drive.ACT.FBK.SeqCamStatus.BothMapc_IP := FALSE;
   RotaryExtractor.Drive.ACT.FBK.SeqCamStatus.SlaveFwd := FALSE;
   RotaryExtractor.Drive.ACT.FBK.SeqCamStatus.SlaveBwd := FALSE;
   RotaryExtractor.Drive.ACT.FBK.SeqCamStatus.SlaveUnwind := FALSE;
   RotaryExtractor.Drive.ACT.FBK.SeqCamStatus.WaitValidByOpe := FALSE;
   RotaryExtractor.Drive.ACT.FBK.SeqCamStatus.MapcA_IP := FALSE;
   RotaryExtractor.Drive.ACT.FBK.SeqCamStatus.MapcB_IP := FALSE;
   RotaryExtractor.Drive.ACT.FBK.SeqCamStatus.MapcC_IP := FALSE;
   RotaryExtractor.Drive.ACT.FBK.SeqCamStatus.CamOnce_PC := FALSE;
   RotaryExtractor.Drive.ACT.FBK.SeqCamStatus.MaxDevError := FALSE;
   RotaryExtractor.Drive.ACT.FBK.SeqCamStatus.PositionCamLockStatus := FALSE;
   RotaryExtractor.Drive.ACT.FBK.SeqCamStatus.WaitRestart := FALSE;
   RotaryExtractor.Drive.ACT.FBK.SeqCamStatus.Bit17 := FALSE;
   RotaryExtractor.Drive.ACT.FBK.SeqCamStatus.Bit18 := FALSE;
   RotaryExtractor.Drive.ACT.FBK.SeqCamStatus.Bit19 := FALSE;
   RotaryExtractor.Drive.ACT.FBK.SeqCamStatus.Bit20 := FALSE;
   RotaryExtractor.Drive.ACT.FBK.SeqCamStatus.Bit21 := FALSE;
   RotaryExtractor.Drive.ACT.FBK.SeqCamStatus.Bit22 := FALSE;
   RotaryExtractor.Drive.ACT.FBK.SeqCamStatus.Bit23 := FALSE;
   RotaryExtractor.Drive.ACT.FBK.SeqCamStatus.Bit24 := FALSE;
   RotaryExtractor.Drive.ACT.FBK.SeqCamStatus.Bit25 := FALSE;
   RotaryExtractor.Drive.ACT.FBK.SeqCamStatus.Bit26 := FALSE;
   RotaryExtractor.Drive.ACT.FBK.SeqCamStatus.Bit27 := FALSE;
   RotaryExtractor.Drive.ACT.FBK.SeqCamStatus.Bit28 := FALSE;
   RotaryExtractor.Drive.ACT.FBK.SeqCamStatus.Bit29 := FALSE;
   RotaryExtractor.Drive.ACT.FBK.SeqCamStatus.Bit30 := FALSE;
   RotaryExtractor.Drive.ACT.FBK.SeqCamStatus.Bit31 := FALSE;
   RotaryExtractor.Drive.ACT.FBK.SeqCamStatus.Bit32 := FALSE;
   RotaryExtractor.Drive.PLS.FinePosOk.LowLimit := 119.0;
   RotaryExtractor.Drive.PLS.FinePosOk.HighLimit := 1.0;
   RotaryExtractor.Drive.PLS.FinePosOk.Ok := TRUE;
   RotaryExtractor.Drive.PLS.KeepPosOk.LowLimit := 0.0;
   RotaryExtractor.Drive.PLS.KeepPosOk.HighLimit := 0.0;
   RotaryExtractor.Drive.PLS.KeepPosOk.Ok := FALSE;
   RotaryExtractor.Drive.PLS.Up.LowLimit := 0.0;
   RotaryExtractor.Drive.PLS.Up.HighLimit := 0.0;
   RotaryExtractor.Drive.PLS.Up.Ok := FALSE;
   RotaryExtractor.Drive.PLS.Intermediate.LowLimit := 0.0;
   RotaryExtractor.Drive.PLS.Intermediate.HighLimit := 0.0;
   RotaryExtractor.Drive.PLS.Intermediate.Ok := FALSE;
   RotaryExtractor.Drive.PLS.Down.LowLimit := 0.0;
   RotaryExtractor.Drive.PLS.Down.HighLimit := 0.0;
   RotaryExtractor.Drive.PLS.Down.Ok := FALSE;
   RotaryExtractor.Drive.PLS.Forward.LowLimit := 0.0;
   RotaryExtractor.Drive.PLS.Forward.HighLimit := 0.0;
   RotaryExtractor.Drive.PLS.Forward.Ok := FALSE;
   RotaryExtractor.Drive.PLS.Backward.LowLimit := 0.0;
   RotaryExtractor.Drive.PLS.Backward.HighLimit := 0.0;
   RotaryExtractor.Drive.PLS.Backward.Ok := FALSE;
   RotaryExtractor.Drive.PLS.Open.LowLimit := 0.0;
   RotaryExtractor.Drive.PLS.Open.HighLimit := 0.0;
   RotaryExtractor.Drive.PLS.Open.Ok := FALSE;
   RotaryExtractor.Drive.PLS.Close.LowLimit := 0.0;
   RotaryExtractor.Drive.PLS.Close.HighLimit := 0.0;
   RotaryExtractor.Drive.PLS.Close.Ok := FALSE;
   RotaryExtractor.Drive.PLS.PreOpen.LowLimit := 0.0;
   RotaryExtractor.Drive.PLS.PreOpen.HighLimit := 0.0;
   RotaryExtractor.Drive.PLS.PreOpen.Ok := FALSE;
   RotaryExtractor.Drive.PLS.Maintenance.LowLimit := 0.0;
   RotaryExtractor.Drive.PLS.Maintenance.HighLimit := 0.0;
   RotaryExtractor.Drive.PLS.Maintenance.Ok := FALSE;
   RotaryExtractor.Drive.PLS.OperatorSide.LowLimit := 0.0;
   RotaryExtractor.Drive.PLS.OperatorSide.HighLimit := 0.0;
   RotaryExtractor.Drive.PLS.OperatorSide.Ok := FALSE;
   RotaryExtractor.Drive.PLS.NotOperatorSide.LowLimit := 0.0;
   RotaryExtractor.Drive.PLS.NotOperatorSide.HighLimit := 0.0;
   RotaryExtractor.Drive.PLS.NotOperatorSide.Ok := FALSE;
   RotaryExtractor.Drive.PLS.OnMould.LowLimit := 0.0;
   RotaryExtractor.Drive.PLS.OnMould.HighLimit := 0.0;
   RotaryExtractor.Drive.PLS.OnMould.Ok := FALSE;
   RotaryExtractor.Drive.PLS.OffMould.LowLimit := 0.0;
   RotaryExtractor.Drive.PLS.OffMould.HighLimit := 0.0;
   RotaryExtractor.Drive.PLS.OffMould.Ok := FALSE;
   RotaryExtractor.Drive.PLS.Pos0.LowLimit := 60.0;
   RotaryExtractor.Drive.PLS.Pos0.HighLimit := 120.1;
   RotaryExtractor.Drive.PLS.Pos0.Ok := FALSE;
   RotaryExtractor.Drive.PLS.Pos1.LowLimit := 0.0;
   RotaryExtractor.Drive.PLS.Pos1.HighLimit := 0.0;
   RotaryExtractor.Drive.PLS.Pos1.Ok := FALSE;
   RotaryExtractor.Drive.PLS.Pos2.LowLimit := 0.0;
   RotaryExtractor.Drive.PLS.Pos2.HighLimit := 0.0;
   RotaryExtractor.Drive.PLS.Pos2.Ok := FALSE;
   RotaryExtractor.Drive.PLS.Pos3.LowLimit := 0.0;
   RotaryExtractor.Drive.PLS.Pos3.HighLimit := 0.0;
   RotaryExtractor.Drive.PLS.Pos3.Ok := FALSE;
   RotaryExtractor.Drive.PLS.Pos4.LowLimit := 0.0;
   RotaryExtractor.Drive.PLS.Pos4.HighLimit := 0.0;
   RotaryExtractor.Drive.PLS.Pos4.Ok := FALSE;
   RotaryExtractor.Drive.PLS.Pos5.LowLimit := 0.0;
   RotaryExtractor.Drive.PLS.Pos5.HighLimit := 0.0;
   RotaryExtractor.Drive.PLS.Pos5.Ok := FALSE;
   RotaryExtractor.Drive.TON_EnableDrive.PT := T#500MS;
   RotaryExtractor.Drive.TON_EnableDrive.IN := FALSE;
   RotaryExtractor.Drive.TON_HwOvertravel_Dis.PT := T#0MS;
   RotaryExtractor.Drive.TON_HwOvertravel_Dis.IN := FALSE;
   RotaryExtractor.Drive.TON_HwOvertravel_En.PT := T#0MS;
   RotaryExtractor.Drive.TON_HwOvertravel_En.IN := FALSE;
   RotaryExtractor.Drive.TON_TimeoutMovement.PT := T#8S;
   RotaryExtractor.Drive.TON_TimeoutMovement.IN := FALSE;
   RotaryExtractor.TON_ResetMaxLevel.PT := T#2S;
   RotaryExtractor.TON_ResetMaxLevel.ET := T#2S;
   RotaryExtractor.TON_ResetMaxLevel.IN := TRUE;
   RotaryExtractor.TON_ResetMaxLevel.Q := TRUE;
   RotaryExtractor.RTO_Work.PT := T#1M;
   RotaryExtractor.RTO_Work.IN := FALSE;
   RotaryExtractor.TON_ScOK.PT := T#20S;
   RotaryExtractor.TON_ScOK.IN := FALSE;
   RotaryExtractor.TON_Sign_MaxLevel.PT := T#1S;
   RotaryExtractor.TON_Sign_MaxLevel.IN := FALSE;
   RotaryExtractor.TON_TimeoutWork.PT := T#20S;
   RotaryExtractor.TON_TimeoutWork.IN := FALSE;
   PickExtractor.ScOk := FALSE;
   PickExtractor.CycleOn := FALSE;
   PickExtractor.Work := FALSE;
   PickExtractor.OkToStop := FALSE;
   PickExtractor.AlmOk := TRUE;
   PickExtractor.DrivesEnabled := FALSE;
   PickExtractor.OutChainObstruction := FALSE;
   PickExtractor.SingleCycle := FALSE;
   PickExtractor.RepositioningReq := FALSE;
   PickExtractor.Ons_TimeWork := FALSE;
   PickExtractor.NumMaxLevel := 0;
   PickExtractor.Input.EnaSel := FALSE;
   PickExtractor.Input.MaxLvl := FALSE;
   PickExtractor.Input.HldOpnNotOpeSid := FALSE;
   PickExtractor.Input.HldClsNotOpeSid := FALSE;
   PickExtractor.Input.HldOpnOpeSid := FALSE;
   PickExtractor.Input.HldClsOpeSid := FALSE;
   PickExtractor.Output.EnaSelLgh := FALSE;
   PickExtractor.Output.HldOpnNotOpeSid := FALSE;
   PickExtractor.Output.HldClsNotOpeSid := FALSE;
   PickExtractor.Output.HldOpnOpeSid := FALSE;
   PickExtractor.Output.HldClsOpeSid := FALSE;
   PickExtractor.Man.Ons_SingleCycle := FALSE;
   PickExtractor.Man.CmdSupportOpen := FALSE;
   PickExtractor.Man.CmdSupportClose := FALSE;
   PickExtractor.Man.CmdSingleCycle := FALSE;
   PickExtractor.Man.EnaPbt := FALSE;
   PickExtractor.Man.RstCmd := FALSE;
   PickExtractor.Man.ScreenNumber := 302_050_301;
   PickExtractor.Man.WithinScreenRange := 0;
   PickExtractor."Step"._00_CycleActived_IntermediateCmd := FALSE;
   PickExtractor."Step"._10_IntermediatePos_OpenSupportCmd := FALSE;
   PickExtractor."Step"._20_OpenSupportPos_DownCmd := FALSE;
   PickExtractor."Step"._30_DownPos_CloseSupportCmd := FALSE;
   PickExtractor."Step"._40_CloseSupportPos_CycleEnd := FALSE;
   PickExtractor."Step".Ons_StrobeWorkDone := FALSE;
   PickExtractor."Step".StrobeWorkDone := FALSE;
   PickExtractor."Step".ScSeqOk := FALSE;
   PickExtractor."Step".SeqActive := FALSE;
   PickExtractor.Drive.AlmOk := FALSE;
   PickExtractor.Drive.AlmEmerg := FALSE;
   PickExtractor.Drive.AlmNode := FALSE;
   PickExtractor.Drive.InitPosDrive := FALSE;
   PickExtractor.Drive.InitPosDrivePLS := FALSE;
   PickExtractor.Drive.GearingON := FALSE;
   PickExtractor.Drive.CamHook := FALSE;
   PickExtractor.Drive.CamStoppingPhase := FALSE;
   PickExtractor.Drive.RepositioningRequest := FALSE;
   PickExtractor.Drive.CamRequestResult := FALSE;
   PickExtractor.Drive.CamRequestError := FALSE;
   PickExtractor.Drive.CamRequestOk := FALSE;
   PickExtractor.Drive.CalibDisAxisReq := FALSE;
   PickExtractor.Drive.CalibReq := FALSE;
   PickExtractor.Drive.CalibProcess := FALSE;
   PickExtractor.Drive.HwOvertravelDisReq := FALSE;
   PickExtractor.Drive.HwOvertravelEnReq := FALSE;
   PickExtractor.Drive.AuxCamRequest := FALSE;
   PickExtractor.Drive.TorquePeakEna := FALSE;
   PickExtractor.Drive.Cmd_Repos := FALSE;
   PickExtractor.Drive.Ons_CamRequest := FALSE;
   PickExtractor.Drive.AuxCmdPosition := 0;
   PickExtractor.Drive.Unwind := 0.0;
   PickExtractor.Drive.MaxDev := 0.0;
   PickExtractor.Drive.ReposSpeed := 100.0;
   PickExtractor.Drive.CalcSlaveDifferenceABS := 0.0;
   PickExtractor.Drive.CalcModPosition := 0.0;
   PickExtractor.Drive.CalcSlaveDifference := 0.0;
   PickExtractor.Drive.CalcMinDeltaPos := 0.0;
   PickExtractor.Drive.CalcMaxDeltaPos := 0.0;
   PickExtractor.Drive.CalcHalfPosUnwind := 0.0;
   PickExtractor.Drive.Man.Cmd_PosJog := FALSE;
   PickExtractor.Drive.Man.Cmd_NegJog := FALSE;
   PickExtractor.Drive.Man.Cmd_Step := FALSE;
   PickExtractor.Drive.Man.Cmd_Forward := FALSE;
   PickExtractor.Drive.Man.Cmd_Backward := FALSE;
   PickExtractor.Drive.Man.Cmd_Up := FALSE;
   PickExtractor.Drive.Man.Cmd_Down := FALSE;
   PickExtractor.Drive.Man.Cmd_Intermediate := FALSE;
   PickExtractor.Drive.Man.Cmd_Open := FALSE;
   PickExtractor.Drive.Man.Cmd_Close := FALSE;
   PickExtractor.Drive.Man.Cmd_PreOpen := FALSE;
   PickExtractor.Drive.Man.Cmd_Maintenance := FALSE;
   PickExtractor.Drive.Man.Cmd_OperatorSide := FALSE;
   PickExtractor.Drive.Man.Cmd_NotOperatorSide := FALSE;
   PickExtractor.Drive.Man.Cmd_OnMould := FALSE;
   PickExtractor.Drive.Man.Cmd_OffMould := FALSE;
   PickExtractor.Drive.Man.Cmd_Pos0 := FALSE;
   PickExtractor.Drive.Man.Cmd_Pos1 := FALSE;
   PickExtractor.Drive.Man.Cmd_Pos2 := FALSE;
   PickExtractor.Drive.Man.Cmd_Pos3 := FALSE;
   PickExtractor.Drive.Man.Cmd_Pos4 := FALSE;
   PickExtractor.Drive.Man.Cmd_Pos5 := FALSE;
   PickExtractor.Drive.Man.Ons_Step := FALSE;
   PickExtractor.Drive.Man.PhaseJogCmd := FALSE;
   PickExtractor.Drive.Man.CmdStartStep := FALSE;
   PickExtractor.Drive.Man.CmdEndStep := FALSE;
   PickExtractor.Drive.Man.StepCond := FALSE;
   PickExtractor.Drive.Man.TON_DelayHomeCmd.PT := T#3S;
   PickExtractor.Drive.Man.TON_DelayHomeCmd.IN := FALSE;
   PickExtractor.Drive.Auto.Cmd_Step := FALSE;
   PickExtractor.Drive.Auto.Cmd_StartStep := FALSE;
   PickExtractor.Drive.Auto.Cmd_EndStep := FALSE;
   PickExtractor.Drive.Auto.Cmd_Forward := FALSE;
   PickExtractor.Drive.Auto.Cmd_Backward := FALSE;
   PickExtractor.Drive.Auto.Cmd_Up := FALSE;
   PickExtractor.Drive.Auto.Cmd_Down := FALSE;
   PickExtractor.Drive.Auto.Cmd_Intermediate := FALSE;
   PickExtractor.Drive.Auto.Cmd_Open := FALSE;
   PickExtractor.Drive.Auto.Cmd_Close := FALSE;
   PickExtractor.Drive.Auto.Cmd_PreOpen := FALSE;
   PickExtractor.Drive.Auto.Cmd_Maintenance := FALSE;
   PickExtractor.Drive.Auto.Cmd_OperatorSide := FALSE;
   PickExtractor.Drive.Auto.Cmd_NotOperatorSide := FALSE;
   PickExtractor.Drive.Auto.Cmd_OnMould := FALSE;
   PickExtractor.Drive.Auto.Cmd_OffMould := FALSE;
   PickExtractor.Drive.Auto.Cmd_Pos0 := FALSE;
   PickExtractor.Drive.Auto.Cmd_Pos1 := FALSE;
   PickExtractor.Drive.Auto.Cmd_Pos2 := FALSE;
   PickExtractor.Drive.Auto.Cmd_Pos3 := FALSE;
   PickExtractor.Drive.Auto.Cmd_Pos4 := FALSE;
   PickExtractor.Drive.Auto.Cmd_Pos5 := FALSE;
   PickExtractor.Drive.Auto.Cmd_Gear := FALSE;
   PickExtractor.Drive.ACT.CMD.Enable := FALSE;
   PickExtractor.Drive.ACT.CMD.Pos_Mode := FALSE;
   PickExtractor.Drive.ACT.CMD.MergeDisabled := FALSE;
   PickExtractor.Drive.ACT.CMD.SCurve := FALSE;
   PickExtractor.Drive.ACT.CMD.Cam_Mode := FALSE;
   PickExtractor.Drive.ACT.CMD.Cam_Request := FALSE;
   PickExtractor.Drive.ACT.CMD.Cam_PhaseStop := FALSE;
   PickExtractor.Drive.ACT.CMD.Gear_Mode := FALSE;
   PickExtractor.Drive.ACT.CMD.Repos_Req := FALSE;
   PickExtractor.Drive.ACT.CMD.Jog_Pos := FALSE;
   PickExtractor.Drive.ACT.CMD.Jog_Neg := FALSE;
   PickExtractor.Drive.ACT.CMD.Stop := FALSE;
   PickExtractor.Drive.ACT.CMD.Calibration_Req := FALSE;
   PickExtractor.Drive.ACT.CMD.Reset := FALSE;
   PickExtractor.Drive.ACT.CMD.RegInput1 := FALSE;
   PickExtractor.Drive.ACT.CMD.Brake_Release := FALSE;
   PickExtractor.Drive.ACT.CMD.HwPosOvertravel_Dis := FALSE;
   PickExtractor.Drive.ACT.CMD.HwNegOvertravel_Dis := FALSE;
   PickExtractor.Drive.ACT.CMD.HwOvertravel_MSG_En := FALSE;
   PickExtractor.Drive.ACT.CMD.OneShootMove := FALSE;
   PickExtractor.Drive.ACT.CMD.Move_Type := 0;
   PickExtractor.Drive.ACT.CMD.Target_Pos := 0.0;
   PickExtractor.Drive.ACT.CMD.Speed := 0.0;
   PickExtractor.Drive.ACT.CMD.Acceleration := 0.0;
   PickExtractor.Drive.ACT.CMD.Deceleration := 0.0;
   PickExtractor.Drive.ACT.CMD.Torque_Limit := 0.0;
   PickExtractor.Drive.ACT.CMD.Gear_Ratio := 0.0;
   PickExtractor.Drive.ACT.CMD.Mccp_Length := 0;
   PickExtractor.Drive.ACT.CMD.Mccp_StartSlope := 0.0;
   PickExtractor.Drive.ACT.CMD.Mccp_EndSlope := 0.0;
   PickExtractor.Drive.ACT.CMD.Mapc_Direction := 0;
   PickExtractor.Drive.ACT.CMD.Mapc_SlaveScaling := 0.0;
   PickExtractor.Drive.ACT.CMD.Mapc_MasterScaling := 0.0;
   PickExtractor.Drive.ACT.CMD.Mapc_MasterLockPosition := 0.0;
   PickExtractor.Drive.ACT.CMD.Mapc_CamLockPosition := 0.0;
   PickExtractor.Drive.ACT.CMD.Cam[0..39].leadingValueStart := 0.0;
   PickExtractor.Drive.ACT.CMD.Cam[0..39].leadingValueEnd := 0.0;
   PickExtractor.Drive.ACT.CMD.Cam[0..39].followingValueStart := 0.0;
   PickExtractor.Drive.ACT.CMD.Cam[0..39].followingValueEnd := 0.0;
   PickExtractor.Drive.ACT.CMD.Cam[0..39].geoVeloStart := 0.0;
   PickExtractor.Drive.ACT.CMD.Cam[0..39].geoVeloEnd := 0.0;
   PickExtractor.Drive.ACT.CMD.Cam[0..39].geoAccelStart := 0.0;
   PickExtractor.Drive.ACT.CMD.Cam[0..39].geoAccelEnd := 0.0;
   PickExtractor.Drive.ACT.CMD.Cam[0..39].geoJerkStart := 0.0;
   PickExtractor.Drive.ACT.CMD.Cam[0..39].geoJerkEnd := 0.0;
   PickExtractor.Drive.ACT.CMD.Cam[0..39].inflectionPointParameter := 0.5;
   PickExtractor.Drive.ACT.CMD.Cam[0..39].modVeloTrapezoidParameter := 1.0;
   PickExtractor.Drive.ACT.CMD.Cam[0..39].modSineMaxAccelCaStar := 0.0;
   PickExtractor.Drive.ACT.CMD.Cam[0..39].camProfileType := 0;
   PickExtractor.Drive.ACT.FBK.Ready := FALSE;
   PickExtractor.Drive.ACT.FBK.Calibrated := FALSE;
   PickExtractor.Drive.ACT.FBK.Fault := FALSE;
   PickExtractor.Drive.ACT.FBK.ModuleConnFault := FALSE;
   PickExtractor.Drive.ACT.FBK.In_Position := FALSE;
   PickExtractor.Drive.ACT.FBK.Standstill := FALSE;
   PickExtractor.Drive.ACT.FBK.Enabled := FALSE;
   PickExtractor.Drive.ACT.FBK.BusReadyStatus := FALSE;
   PickExtractor.Drive.ACT.FBK.BrakeReleased := FALSE;
   PickExtractor.Drive.ACT.FBK.HwPosOvertravelDisabled := FALSE;
   PickExtractor.Drive.ACT.FBK.HwNegOvertravelDisabled := FALSE;
   PickExtractor.Drive.ACT.FBK.SafeOffStatus := FALSE;
   PickExtractor.Drive.ACT.FBK.MaxTorqueLimit := FALSE;
   PickExtractor.Drive.ACT.FBK.PosMerge_IP := FALSE;
   PickExtractor.Drive.ACT.FBK.PosMerge_PC := FALSE;
   PickExtractor.Drive.ACT.FBK.Gearing_IP := FALSE;
   PickExtractor.Drive.ACT.FBK.Position := 0.0;
   PickExtractor.Drive.ACT.FBK.Speed := 0.0;
   PickExtractor.Drive.ACT.FBK.Torque := 0.0;
   PickExtractor.Drive.ACT.FBK.RegInput1Pos := 0.0;
   PickExtractor.Drive.ACT.FBK.SeqCamErrorCode := 0;
   PickExtractor.Drive.ACT.FBK.SeqCamTargetPosMAM := 0.0;
   PickExtractor.Drive.ACT.FBK.SeqCamStatus.EndSequence := FALSE;
   PickExtractor.Drive.ACT.FBK.SeqCamStatus.EndSuccess := FALSE;
   PickExtractor.Drive.ACT.FBK.SeqCamStatus.EndError := FALSE;
   PickExtractor.Drive.ACT.FBK.SeqCamStatus.CamHook := FALSE;
   PickExtractor.Drive.ACT.FBK.SeqCamStatus.BothMapc_IP := FALSE;
   PickExtractor.Drive.ACT.FBK.SeqCamStatus.SlaveFwd := FALSE;
   PickExtractor.Drive.ACT.FBK.SeqCamStatus.SlaveBwd := FALSE;
   PickExtractor.Drive.ACT.FBK.SeqCamStatus.SlaveUnwind := FALSE;
   PickExtractor.Drive.ACT.FBK.SeqCamStatus.WaitValidByOpe := FALSE;
   PickExtractor.Drive.ACT.FBK.SeqCamStatus.MapcA_IP := FALSE;
   PickExtractor.Drive.ACT.FBK.SeqCamStatus.MapcB_IP := FALSE;
   PickExtractor.Drive.ACT.FBK.SeqCamStatus.MapcC_IP := FALSE;
   PickExtractor.Drive.ACT.FBK.SeqCamStatus.CamOnce_PC := FALSE;
   PickExtractor.Drive.ACT.FBK.SeqCamStatus.MaxDevError := FALSE;
   PickExtractor.Drive.ACT.FBK.SeqCamStatus.PositionCamLockStatus := FALSE;
   PickExtractor.Drive.ACT.FBK.SeqCamStatus.WaitRestart := FALSE;
   PickExtractor.Drive.ACT.FBK.SeqCamStatus.Bit17 := FALSE;
   PickExtractor.Drive.ACT.FBK.SeqCamStatus.Bit18 := FALSE;
   PickExtractor.Drive.ACT.FBK.SeqCamStatus.Bit19 := FALSE;
   PickExtractor.Drive.ACT.FBK.SeqCamStatus.Bit20 := FALSE;
   PickExtractor.Drive.ACT.FBK.SeqCamStatus.Bit21 := FALSE;
   PickExtractor.Drive.ACT.FBK.SeqCamStatus.Bit22 := FALSE;
   PickExtractor.Drive.ACT.FBK.SeqCamStatus.Bit23 := FALSE;
   PickExtractor.Drive.ACT.FBK.SeqCamStatus.Bit24 := FALSE;
   PickExtractor.Drive.ACT.FBK.SeqCamStatus.Bit25 := FALSE;
   PickExtractor.Drive.ACT.FBK.SeqCamStatus.Bit26 := FALSE;
   PickExtractor.Drive.ACT.FBK.SeqCamStatus.Bit27 := FALSE;
   PickExtractor.Drive.ACT.FBK.SeqCamStatus.Bit28 := FALSE;
   PickExtractor.Drive.ACT.FBK.SeqCamStatus.Bit29 := FALSE;
   PickExtractor.Drive.ACT.FBK.SeqCamStatus.Bit30 := FALSE;
   PickExtractor.Drive.ACT.FBK.SeqCamStatus.Bit31 := FALSE;
   PickExtractor.Drive.ACT.FBK.SeqCamStatus.Bit32 := FALSE;
   PickExtractor.Drive.PLS.FinePosOk.LowLimit := 0.0;
   PickExtractor.Drive.PLS.FinePosOk.HighLimit := 0.0;
   PickExtractor.Drive.PLS.FinePosOk.Ok := FALSE;
   PickExtractor.Drive.PLS.KeepPosOk.LowLimit := 0.0;
   PickExtractor.Drive.PLS.KeepPosOk.HighLimit := 0.0;
   PickExtractor.Drive.PLS.KeepPosOk.Ok := FALSE;
   PickExtractor.Drive.PLS.Up.LowLimit := 0.0;
   PickExtractor.Drive.PLS.Up.HighLimit := 0.0;
   PickExtractor.Drive.PLS.Up.Ok := FALSE;
   PickExtractor.Drive.PLS.Intermediate.LowLimit := 0.0;
   PickExtractor.Drive.PLS.Intermediate.HighLimit := 0.0;
   PickExtractor.Drive.PLS.Intermediate.Ok := FALSE;
   PickExtractor.Drive.PLS.Down.LowLimit := 0.0;
   PickExtractor.Drive.PLS.Down.HighLimit := 0.0;
   PickExtractor.Drive.PLS.Down.Ok := FALSE;
   PickExtractor.Drive.PLS.Forward.LowLimit := 0.0;
   PickExtractor.Drive.PLS.Forward.HighLimit := 0.0;
   PickExtractor.Drive.PLS.Forward.Ok := FALSE;
   PickExtractor.Drive.PLS.Backward.LowLimit := 0.0;
   PickExtractor.Drive.PLS.Backward.HighLimit := 0.0;
   PickExtractor.Drive.PLS.Backward.Ok := FALSE;
   PickExtractor.Drive.PLS.Open.LowLimit := 0.0;
   PickExtractor.Drive.PLS.Open.HighLimit := 0.0;
   PickExtractor.Drive.PLS.Open.Ok := FALSE;
   PickExtractor.Drive.PLS.Close.LowLimit := 0.0;
   PickExtractor.Drive.PLS.Close.HighLimit := 0.0;
   PickExtractor.Drive.PLS.Close.Ok := FALSE;
   PickExtractor.Drive.PLS.PreOpen.LowLimit := 0.0;
   PickExtractor.Drive.PLS.PreOpen.HighLimit := 0.0;
   PickExtractor.Drive.PLS.PreOpen.Ok := FALSE;
   PickExtractor.Drive.PLS.Maintenance.LowLimit := 0.0;
   PickExtractor.Drive.PLS.Maintenance.HighLimit := 0.0;
   PickExtractor.Drive.PLS.Maintenance.Ok := FALSE;
   PickExtractor.Drive.PLS.OperatorSide.LowLimit := 0.0;
   PickExtractor.Drive.PLS.OperatorSide.HighLimit := 0.0;
   PickExtractor.Drive.PLS.OperatorSide.Ok := FALSE;
   PickExtractor.Drive.PLS.NotOperatorSide.LowLimit := 0.0;
   PickExtractor.Drive.PLS.NotOperatorSide.HighLimit := 0.0;
   PickExtractor.Drive.PLS.NotOperatorSide.Ok := FALSE;
   PickExtractor.Drive.PLS.OnMould.LowLimit := 0.0;
   PickExtractor.Drive.PLS.OnMould.HighLimit := 0.0;
   PickExtractor.Drive.PLS.OnMould.Ok := FALSE;
   PickExtractor.Drive.PLS.OffMould.LowLimit := 0.0;
   PickExtractor.Drive.PLS.OffMould.HighLimit := 0.0;
   PickExtractor.Drive.PLS.OffMould.Ok := FALSE;
   PickExtractor.Drive.PLS.Pos0.LowLimit := 0.0;
   PickExtractor.Drive.PLS.Pos0.HighLimit := 0.0;
   PickExtractor.Drive.PLS.Pos0.Ok := FALSE;
   PickExtractor.Drive.PLS.Pos1.LowLimit := 0.0;
   PickExtractor.Drive.PLS.Pos1.HighLimit := 0.0;
   PickExtractor.Drive.PLS.Pos1.Ok := FALSE;
   PickExtractor.Drive.PLS.Pos2.LowLimit := 0.0;
   PickExtractor.Drive.PLS.Pos2.HighLimit := 0.0;
   PickExtractor.Drive.PLS.Pos2.Ok := FALSE;
   PickExtractor.Drive.PLS.Pos3.LowLimit := 0.0;
   PickExtractor.Drive.PLS.Pos3.HighLimit := 0.0;
   PickExtractor.Drive.PLS.Pos3.Ok := FALSE;
   PickExtractor.Drive.PLS.Pos4.LowLimit := 0.0;
   PickExtractor.Drive.PLS.Pos4.HighLimit := 0.0;
   PickExtractor.Drive.PLS.Pos4.Ok := FALSE;
   PickExtractor.Drive.PLS.Pos5.LowLimit := 0.0;
   PickExtractor.Drive.PLS.Pos5.HighLimit := 0.0;
   PickExtractor.Drive.PLS.Pos5.Ok := FALSE;
   PickExtractor.Drive.TON_EnableDrive.PT := T#500MS;
   PickExtractor.Drive.TON_EnableDrive.IN := FALSE;
   PickExtractor.Drive.TON_HwOvertravel_Dis.PT := T#0MS;
   PickExtractor.Drive.TON_HwOvertravel_Dis.IN := FALSE;
   PickExtractor.Drive.TON_HwOvertravel_En.PT := T#0MS;
   PickExtractor.Drive.TON_HwOvertravel_En.IN := FALSE;
   PickExtractor.Drive.TON_TimeoutMovement.PT := T#8S;
   PickExtractor.Drive.TON_TimeoutMovement.IN := FALSE;
   PickExtractor.TON_ResetMaxLevel.PT := T#2S;
   PickExtractor.TON_ResetMaxLevel.IN := FALSE;
   PickExtractor.RTO_Work.PT := T#1M;
   PickExtractor.RTO_Work.IN := FALSE;
   PickExtractor.TON_ScOK.PT := T#20S;
   PickExtractor.TON_ScOK.IN := FALSE;
   PickExtractor.TON_IncorrectPosOpeSide.PT := T#4S;
   PickExtractor.TON_IncorrectPosOpeSide.IN := FALSE;
   PickExtractor.TON_IncorrectPosNotOpeSide.PT := T#4S;
   PickExtractor.TON_IncorrectPosNotOpeSide.IN := FALSE;
   PickExtractor.TON_Sign_MaxLevel.PT := T#1S;
   PickExtractor.TON_Sign_MaxLevel.IN := FALSE;
   PickExtractor.TON_TimeoutWork.PT := T#20S;
   PickExtractor.TON_TimeoutWork.IN := FALSE;
   BookedExtractor.ScOk := FALSE;
   BookedExtractor.CycleOn := FALSE;
   BookedExtractor.Work := FALSE;
   BookedExtractor.OkToStop := TRUE;
   BookedExtractor.AlmOk := TRUE;
   BookedExtractor.DrivesEnabled := FALSE;
   BookedExtractor.OutChainObstruction := TRUE;
   BookedExtractor.SingleCycle := FALSE;
   BookedExtractor.RepositioningReq := FALSE;
   BookedExtractor.Ons_TimeWork := TRUE;
   BookedExtractor.NumMaxLevel := 0;
   BookedExtractor.Input.EnaSel := FALSE;
   BookedExtractor.Input.MaxLvl := FALSE;
   BookedExtractor.Input.HldOpnNotOpeSid := FALSE;
   BookedExtractor.Input.HldClsNotOpeSid := TRUE;
   BookedExtractor.Input.HldOpnOpeSid := FALSE;
   BookedExtractor.Input.HldClsOpeSid := TRUE;
   BookedExtractor.Input.HigProMou := FALSE;
   BookedExtractor.Output.EnaSelLgh := FALSE;
   BookedExtractor.Output.HldOpnNotOpeSid := FALSE;
   BookedExtractor.Output.HldClsNotOpeSid := FALSE;
   BookedExtractor.Output.HldOpnOpeSid := FALSE;
   BookedExtractor.Output.HldClsOpeSid := FALSE;
   BookedExtractor.Man.Ons_SingleCycle := FALSE;
   BookedExtractor.Man.CmdSupportOpen := FALSE;
   BookedExtractor.Man.CmdSupportClose := FALSE;
   BookedExtractor.Man.CmdSingleCycle := FALSE;
   BookedExtractor.Man.EnaPbt := FALSE;
   BookedExtractor.Man.RstCmd := TRUE;
   BookedExtractor.Man.ScreenNumber := 302_060_301;
   BookedExtractor.Man.WithinScreenRange := 0;
   BookedExtractor."Step"._00_CycleActived_UpCmd := FALSE;
   BookedExtractor."Step"._10_PickUpPos_StoreStepCmd := FALSE;
   BookedExtractor."Step"._20_StepInMotion_PickIntermediateCmd := FALSE;
   BookedExtractor."Step"._25_StoreStepDone := FALSE;
   BookedExtractor."Step"._30_PickIntermediatePos_OpenSupportCmd := FALSE;
   BookedExtractor."Step"._40_OpenSupportPos_PickDownCmd := FALSE;
   BookedExtractor."Step"._50_PickDownPos_CloseSupportCmd := FALSE;
   BookedExtractor."Step"._60_CloseSupportPos_CycleEnd := FALSE;
   BookedExtractor."Step".Ons_StrobeWorkDone := FALSE;
   BookedExtractor."Step".StrobeWorkDone := FALSE;
   BookedExtractor."Step".ScSeqOk := FALSE;
   BookedExtractor."Step".SeqActive := FALSE;
   BookedExtractor.DrivePick.AlmOk := FALSE;
   BookedExtractor.DrivePick.AlmEmerg := FALSE;
   BookedExtractor.DrivePick.AlmNode := FALSE;
   BookedExtractor.DrivePick.InitPosDrive := FALSE;
   BookedExtractor.DrivePick.InitPosDrivePLS := FALSE;
   BookedExtractor.DrivePick.GearingON := FALSE;
   BookedExtractor.DrivePick.CamHook := FALSE;
   BookedExtractor.DrivePick.CamStoppingPhase := FALSE;
   BookedExtractor.DrivePick.RepositioningRequest := FALSE;
   BookedExtractor.DrivePick.CamRequestResult := FALSE;
   BookedExtractor.DrivePick.CamRequestError := FALSE;
   BookedExtractor.DrivePick.CamRequestOk := FALSE;
   BookedExtractor.DrivePick.CalibDisAxisReq := FALSE;
   BookedExtractor.DrivePick.CalibReq := FALSE;
   BookedExtractor.DrivePick.CalibProcess := FALSE;
   BookedExtractor.DrivePick.HwOvertravelDisReq := FALSE;
   BookedExtractor.DrivePick.HwOvertravelEnReq := FALSE;
   BookedExtractor.DrivePick.AuxCamRequest := FALSE;
   BookedExtractor.DrivePick.TorquePeakEna := TRUE;
   BookedExtractor.DrivePick.Cmd_Repos := FALSE;
   BookedExtractor.DrivePick.Ons_CamRequest := FALSE;
   BookedExtractor.DrivePick.AuxCmdPosition := 0;
   BookedExtractor.DrivePick.Unwind := 0.0;
   BookedExtractor.DrivePick.MaxDev := 0.0;
   BookedExtractor.DrivePick.ReposSpeed := 100.0;
   BookedExtractor.DrivePick.CalcSlaveDifferenceABS := 0.0;
   BookedExtractor.DrivePick.CalcModPosition := 0.0;
   BookedExtractor.DrivePick.CalcSlaveDifference := 0.0;
   BookedExtractor.DrivePick.CalcMinDeltaPos := 0.0;
   BookedExtractor.DrivePick.CalcMaxDeltaPos := 0.0;
   BookedExtractor.DrivePick.CalcHalfPosUnwind := 0.0;
   BookedExtractor.DrivePick.Man.Cmd_PosJog := FALSE;
   BookedExtractor.DrivePick.Man.Cmd_NegJog := FALSE;
   BookedExtractor.DrivePick.Man.Cmd_Step := FALSE;
   BookedExtractor.DrivePick.Man.Cmd_Forward := FALSE;
   BookedExtractor.DrivePick.Man.Cmd_Backward := FALSE;
   BookedExtractor.DrivePick.Man.Cmd_Up := FALSE;
   BookedExtractor.DrivePick.Man.Cmd_Down := FALSE;
   BookedExtractor.DrivePick.Man.Cmd_Intermediate := FALSE;
   BookedExtractor.DrivePick.Man.Cmd_Open := FALSE;
   BookedExtractor.DrivePick.Man.Cmd_Close := FALSE;
   BookedExtractor.DrivePick.Man.Cmd_PreOpen := FALSE;
   BookedExtractor.DrivePick.Man.Cmd_Maintenance := FALSE;
   BookedExtractor.DrivePick.Man.Cmd_OperatorSide := FALSE;
   BookedExtractor.DrivePick.Man.Cmd_NotOperatorSide := FALSE;
   BookedExtractor.DrivePick.Man.Cmd_OnMould := FALSE;
   BookedExtractor.DrivePick.Man.Cmd_OffMould := FALSE;
   BookedExtractor.DrivePick.Man.Cmd_Pos0 := FALSE;
   BookedExtractor.DrivePick.Man.Cmd_Pos1 := FALSE;
   BookedExtractor.DrivePick.Man.Cmd_Pos2 := FALSE;
   BookedExtractor.DrivePick.Man.Cmd_Pos3 := FALSE;
   BookedExtractor.DrivePick.Man.Cmd_Pos4 := FALSE;
   BookedExtractor.DrivePick.Man.Cmd_Pos5 := FALSE;
   BookedExtractor.DrivePick.Man.Ons_Step := FALSE;
   BookedExtractor.DrivePick.Man.PhaseJogCmd := FALSE;
   BookedExtractor.DrivePick.Man.CmdStartStep := FALSE;
   BookedExtractor.DrivePick.Man.CmdEndStep := FALSE;
   BookedExtractor.DrivePick.Man.StepCond := FALSE;
   BookedExtractor.DrivePick.Man.TON_DelayHomeCmd.PT := T#3S;
   BookedExtractor.DrivePick.Man.TON_DelayHomeCmd.IN := FALSE;
   BookedExtractor.DrivePick.Auto.Cmd_Step := FALSE;
   BookedExtractor.DrivePick.Auto.Cmd_StartStep := FALSE;
   BookedExtractor.DrivePick.Auto.Cmd_EndStep := FALSE;
   BookedExtractor.DrivePick.Auto.Cmd_Forward := FALSE;
   BookedExtractor.DrivePick.Auto.Cmd_Backward := FALSE;
   BookedExtractor.DrivePick.Auto.Cmd_Up := FALSE;
   BookedExtractor.DrivePick.Auto.Cmd_Down := FALSE;
   BookedExtractor.DrivePick.Auto.Cmd_Intermediate := FALSE;
   BookedExtractor.DrivePick.Auto.Cmd_Open := FALSE;
   BookedExtractor.DrivePick.Auto.Cmd_Close := FALSE;
   BookedExtractor.DrivePick.Auto.Cmd_PreOpen := FALSE;
   BookedExtractor.DrivePick.Auto.Cmd_Maintenance := FALSE;
   BookedExtractor.DrivePick.Auto.Cmd_OperatorSide := FALSE;
   BookedExtractor.DrivePick.Auto.Cmd_NotOperatorSide := FALSE;
   BookedExtractor.DrivePick.Auto.Cmd_OnMould := FALSE;
   BookedExtractor.DrivePick.Auto.Cmd_OffMould := FALSE;
   BookedExtractor.DrivePick.Auto.Cmd_Pos0 := FALSE;
   BookedExtractor.DrivePick.Auto.Cmd_Pos1 := FALSE;
   BookedExtractor.DrivePick.Auto.Cmd_Pos2 := FALSE;
   BookedExtractor.DrivePick.Auto.Cmd_Pos3 := FALSE;
   BookedExtractor.DrivePick.Auto.Cmd_Pos4 := FALSE;
   BookedExtractor.DrivePick.Auto.Cmd_Pos5 := FALSE;
   BookedExtractor.DrivePick.Auto.Cmd_Gear := FALSE;
   BookedExtractor.DrivePick.ACT.CMD.Enable := FALSE;
   BookedExtractor.DrivePick.ACT.CMD.Pos_Mode := FALSE;
   BookedExtractor.DrivePick.ACT.CMD.MergeDisabled := FALSE;
   BookedExtractor.DrivePick.ACT.CMD.SCurve := FALSE;
   BookedExtractor.DrivePick.ACT.CMD.Cam_Mode := FALSE;
   BookedExtractor.DrivePick.ACT.CMD.Cam_Request := FALSE;
   BookedExtractor.DrivePick.ACT.CMD.Cam_PhaseStop := FALSE;
   BookedExtractor.DrivePick.ACT.CMD.Gear_Mode := FALSE;
   BookedExtractor.DrivePick.ACT.CMD.Repos_Req := FALSE;
   BookedExtractor.DrivePick.ACT.CMD.Jog_Pos := FALSE;
   BookedExtractor.DrivePick.ACT.CMD.Jog_Neg := FALSE;
   BookedExtractor.DrivePick.ACT.CMD.Stop := TRUE;
   BookedExtractor.DrivePick.ACT.CMD.Calibration_Req := FALSE;
   BookedExtractor.DrivePick.ACT.CMD.Reset := FALSE;
   BookedExtractor.DrivePick.ACT.CMD.RegInput1 := FALSE;
   BookedExtractor.DrivePick.ACT.CMD.Brake_Release := FALSE;
   BookedExtractor.DrivePick.ACT.CMD.HwPosOvertravel_Dis := FALSE;
   BookedExtractor.DrivePick.ACT.CMD.HwNegOvertravel_Dis := FALSE;
   BookedExtractor.DrivePick.ACT.CMD.HwOvertravel_MSG_En := FALSE;
   BookedExtractor.DrivePick.ACT.CMD.OneShootMove := FALSE;
   BookedExtractor.DrivePick.ACT.CMD.Move_Type := 0;
   BookedExtractor.DrivePick.ACT.CMD.Target_Pos := 2.0;
   BookedExtractor.DrivePick.ACT.CMD.Speed := 100.0;
   BookedExtractor.DrivePick.ACT.CMD.Acceleration := 4000.0;
   BookedExtractor.DrivePick.ACT.CMD.Deceleration := 4500.0;
   BookedExtractor.DrivePick.ACT.CMD.Torque_Limit := 15.0;
   BookedExtractor.DrivePick.ACT.CMD.Gear_Ratio := 0.0;
   BookedExtractor.DrivePick.ACT.CMD.Mccp_Length := 0;
   BookedExtractor.DrivePick.ACT.CMD.Mccp_StartSlope := 0.0;
   BookedExtractor.DrivePick.ACT.CMD.Mccp_EndSlope := 0.0;
   BookedExtractor.DrivePick.ACT.CMD.Mapc_Direction := 0;
   BookedExtractor.DrivePick.ACT.CMD.Mapc_SlaveScaling := 0.0;
   BookedExtractor.DrivePick.ACT.CMD.Mapc_MasterScaling := 0.0;
   BookedExtractor.DrivePick.ACT.CMD.Mapc_MasterLockPosition := 0.0;
   BookedExtractor.DrivePick.ACT.CMD.Mapc_CamLockPosition := 0.0;
   BookedExtractor.DrivePick.ACT.CMD.Cam[0..39].leadingValueStart := 0.0;
   BookedExtractor.DrivePick.ACT.CMD.Cam[0..39].leadingValueEnd := 0.0;
   BookedExtractor.DrivePick.ACT.CMD.Cam[0..39].followingValueStart := 0.0;
   BookedExtractor.DrivePick.ACT.CMD.Cam[0..39].followingValueEnd := 0.0;
   BookedExtractor.DrivePick.ACT.CMD.Cam[0..39].geoVeloStart := 0.0;
   BookedExtractor.DrivePick.ACT.CMD.Cam[0..39].geoVeloEnd := 0.0;
   BookedExtractor.DrivePick.ACT.CMD.Cam[0..39].geoAccelStart := 0.0;
   BookedExtractor.DrivePick.ACT.CMD.Cam[0..39].geoAccelEnd := 0.0;
   BookedExtractor.DrivePick.ACT.CMD.Cam[0..39].geoJerkStart := 0.0;
   BookedExtractor.DrivePick.ACT.CMD.Cam[0..39].geoJerkEnd := 0.0;
   BookedExtractor.DrivePick.ACT.CMD.Cam[0..39].inflectionPointParameter := 0.5;
   BookedExtractor.DrivePick.ACT.CMD.Cam[0..39].modVeloTrapezoidParameter := 1.0;
   BookedExtractor.DrivePick.ACT.CMD.Cam[0..39].modSineMaxAccelCaStar := 0.0;
   BookedExtractor.DrivePick.ACT.CMD.Cam[0..39].camProfileType := 0;
   BookedExtractor.DrivePick.ACT.FBK.Ready := TRUE;
   BookedExtractor.DrivePick.ACT.FBK.Calibrated := TRUE;
   BookedExtractor.DrivePick.ACT.FBK.Fault := FALSE;
   BookedExtractor.DrivePick.ACT.FBK.ModuleConnFault := FALSE;
   BookedExtractor.DrivePick.ACT.FBK.In_Position := FALSE;
   BookedExtractor.DrivePick.ACT.FBK.Standstill := TRUE;
   BookedExtractor.DrivePick.ACT.FBK.Enabled := FALSE;
   BookedExtractor.DrivePick.ACT.FBK.BusReadyStatus := FALSE;
   BookedExtractor.DrivePick.ACT.FBK.BrakeReleased := FALSE;
   BookedExtractor.DrivePick.ACT.FBK.HwPosOvertravelDisabled := FALSE;
   BookedExtractor.DrivePick.ACT.FBK.HwNegOvertravelDisabled := FALSE;
   BookedExtractor.DrivePick.ACT.FBK.SafeOffStatus := FALSE;
   BookedExtractor.DrivePick.ACT.FBK.MaxTorqueLimit := FALSE;
   BookedExtractor.DrivePick.ACT.FBK.PosMerge_IP := FALSE;
   BookedExtractor.DrivePick.ACT.FBK.PosMerge_PC := FALSE;
   BookedExtractor.DrivePick.ACT.FBK.Gearing_IP := FALSE;
   BookedExtractor.DrivePick.ACT.FBK.Position := 1.991;
   BookedExtractor.DrivePick.ACT.FBK.Speed := 0.0;
   BookedExtractor.DrivePick.ACT.FBK.Torque := 0.0;
   BookedExtractor.DrivePick.ACT.FBK.RegInput1Pos := 0.0;
   BookedExtractor.DrivePick.ACT.FBK.SeqCamErrorCode := 0;
   BookedExtractor.DrivePick.ACT.FBK.SeqCamTargetPosMAM := 0.0;
   BookedExtractor.DrivePick.ACT.FBK.SeqCamStatus.EndSequence := FALSE;
   BookedExtractor.DrivePick.ACT.FBK.SeqCamStatus.EndSuccess := FALSE;
   BookedExtractor.DrivePick.ACT.FBK.SeqCamStatus.EndError := FALSE;
   BookedExtractor.DrivePick.ACT.FBK.SeqCamStatus.CamHook := FALSE;
   BookedExtractor.DrivePick.ACT.FBK.SeqCamStatus.BothMapc_IP := FALSE;
   BookedExtractor.DrivePick.ACT.FBK.SeqCamStatus.SlaveFwd := FALSE;
   BookedExtractor.DrivePick.ACT.FBK.SeqCamStatus.SlaveBwd := FALSE;
   BookedExtractor.DrivePick.ACT.FBK.SeqCamStatus.SlaveUnwind := FALSE;
   BookedExtractor.DrivePick.ACT.FBK.SeqCamStatus.WaitValidByOpe := FALSE;
   BookedExtractor.DrivePick.ACT.FBK.SeqCamStatus.MapcA_IP := FALSE;
   BookedExtractor.DrivePick.ACT.FBK.SeqCamStatus.MapcB_IP := FALSE;
   BookedExtractor.DrivePick.ACT.FBK.SeqCamStatus.MapcC_IP := FALSE;
   BookedExtractor.DrivePick.ACT.FBK.SeqCamStatus.CamOnce_PC := FALSE;
   BookedExtractor.DrivePick.ACT.FBK.SeqCamStatus.MaxDevError := FALSE;
   BookedExtractor.DrivePick.ACT.FBK.SeqCamStatus.PositionCamLockStatus := FALSE;
   BookedExtractor.DrivePick.ACT.FBK.SeqCamStatus.WaitRestart := FALSE;
   BookedExtractor.DrivePick.ACT.FBK.SeqCamStatus.Bit17 := FALSE;
   BookedExtractor.DrivePick.ACT.FBK.SeqCamStatus.Bit18 := FALSE;
   BookedExtractor.DrivePick.ACT.FBK.SeqCamStatus.Bit19 := FALSE;
   BookedExtractor.DrivePick.ACT.FBK.SeqCamStatus.Bit20 := FALSE;
   BookedExtractor.DrivePick.ACT.FBK.SeqCamStatus.Bit21 := FALSE;
   BookedExtractor.DrivePick.ACT.FBK.SeqCamStatus.Bit22 := FALSE;
   BookedExtractor.DrivePick.ACT.FBK.SeqCamStatus.Bit23 := FALSE;
   BookedExtractor.DrivePick.ACT.FBK.SeqCamStatus.Bit24 := FALSE;
   BookedExtractor.DrivePick.ACT.FBK.SeqCamStatus.Bit25 := FALSE;
   BookedExtractor.DrivePick.ACT.FBK.SeqCamStatus.Bit26 := FALSE;
   BookedExtractor.DrivePick.ACT.FBK.SeqCamStatus.Bit27 := FALSE;
   BookedExtractor.DrivePick.ACT.FBK.SeqCamStatus.Bit28 := FALSE;
   BookedExtractor.DrivePick.ACT.FBK.SeqCamStatus.Bit29 := FALSE;
   BookedExtractor.DrivePick.ACT.FBK.SeqCamStatus.Bit30 := FALSE;
   BookedExtractor.DrivePick.ACT.FBK.SeqCamStatus.Bit31 := FALSE;
   BookedExtractor.DrivePick.ACT.FBK.SeqCamStatus.Bit32 := FALSE;
   BookedExtractor.DrivePick.PLS.FinePosOk.LowLimit := 0.0;
   BookedExtractor.DrivePick.PLS.FinePosOk.HighLimit := 0.0;
   BookedExtractor.DrivePick.PLS.FinePosOk.Ok := FALSE;
   BookedExtractor.DrivePick.PLS.KeepPosOk.LowLimit := 0.0;
   BookedExtractor.DrivePick.PLS.KeepPosOk.HighLimit := 0.0;
   BookedExtractor.DrivePick.PLS.KeepPosOk.Ok := FALSE;
   BookedExtractor.DrivePick.PLS.Up.LowLimit := 89.0;
   BookedExtractor.DrivePick.PLS.Up.HighLimit := 91.0;
   BookedExtractor.DrivePick.PLS.Up.Ok := FALSE;
   BookedExtractor.DrivePick.PLS.Intermediate.LowLimit := 74.0;
   BookedExtractor.DrivePick.PLS.Intermediate.HighLimit := 76.0;
   BookedExtractor.DrivePick.PLS.Intermediate.Ok := FALSE;
   BookedExtractor.DrivePick.PLS.Down.LowLimit := 1.0;
   BookedExtractor.DrivePick.PLS.Down.HighLimit := 3.0;
   BookedExtractor.DrivePick.PLS.Down.Ok := TRUE;
   BookedExtractor.DrivePick.PLS.Forward.LowLimit := 0.0;
   BookedExtractor.DrivePick.PLS.Forward.HighLimit := 0.0;
   BookedExtractor.DrivePick.PLS.Forward.Ok := FALSE;
   BookedExtractor.DrivePick.PLS.Backward.LowLimit := 0.0;
   BookedExtractor.DrivePick.PLS.Backward.HighLimit := 0.0;
   BookedExtractor.DrivePick.PLS.Backward.Ok := FALSE;
   BookedExtractor.DrivePick.PLS.Open.LowLimit := 0.0;
   BookedExtractor.DrivePick.PLS.Open.HighLimit := 0.0;
   BookedExtractor.DrivePick.PLS.Open.Ok := FALSE;
   BookedExtractor.DrivePick.PLS.Close.LowLimit := 0.0;
   BookedExtractor.DrivePick.PLS.Close.HighLimit := 0.0;
   BookedExtractor.DrivePick.PLS.Close.Ok := FALSE;
   BookedExtractor.DrivePick.PLS.PreOpen.LowLimit := 0.0;
   BookedExtractor.DrivePick.PLS.PreOpen.HighLimit := 0.0;
   BookedExtractor.DrivePick.PLS.PreOpen.Ok := FALSE;
   BookedExtractor.DrivePick.PLS.Maintenance.LowLimit := 0.0;
   BookedExtractor.DrivePick.PLS.Maintenance.HighLimit := 0.0;
   BookedExtractor.DrivePick.PLS.Maintenance.Ok := FALSE;
   BookedExtractor.DrivePick.PLS.OperatorSide.LowLimit := 0.0;
   BookedExtractor.DrivePick.PLS.OperatorSide.HighLimit := 0.0;
   BookedExtractor.DrivePick.PLS.OperatorSide.Ok := FALSE;
   BookedExtractor.DrivePick.PLS.NotOperatorSide.LowLimit := 0.0;
   BookedExtractor.DrivePick.PLS.NotOperatorSide.HighLimit := 0.0;
   BookedExtractor.DrivePick.PLS.NotOperatorSide.Ok := FALSE;
   BookedExtractor.DrivePick.PLS.OnMould.LowLimit := 0.0;
   BookedExtractor.DrivePick.PLS.OnMould.HighLimit := 0.0;
   BookedExtractor.DrivePick.PLS.OnMould.Ok := FALSE;
   BookedExtractor.DrivePick.PLS.OffMould.LowLimit := 0.0;
   BookedExtractor.DrivePick.PLS.OffMould.HighLimit := 0.0;
   BookedExtractor.DrivePick.PLS.OffMould.Ok := FALSE;
   BookedExtractor.DrivePick.PLS.Pos0.LowLimit := 0.0;
   BookedExtractor.DrivePick.PLS.Pos0.HighLimit := 0.0;
   BookedExtractor.DrivePick.PLS.Pos0.Ok := FALSE;
   BookedExtractor.DrivePick.PLS.Pos1.LowLimit := 0.0;
   BookedExtractor.DrivePick.PLS.Pos1.HighLimit := 0.0;
   BookedExtractor.DrivePick.PLS.Pos1.Ok := FALSE;
   BookedExtractor.DrivePick.PLS.Pos2.LowLimit := 0.0;
   BookedExtractor.DrivePick.PLS.Pos2.HighLimit := 0.0;
   BookedExtractor.DrivePick.PLS.Pos2.Ok := FALSE;
   BookedExtractor.DrivePick.PLS.Pos3.LowLimit := 0.0;
   BookedExtractor.DrivePick.PLS.Pos3.HighLimit := 0.0;
   BookedExtractor.DrivePick.PLS.Pos3.Ok := FALSE;
   BookedExtractor.DrivePick.PLS.Pos4.LowLimit := 0.0;
   BookedExtractor.DrivePick.PLS.Pos4.HighLimit := 0.0;
   BookedExtractor.DrivePick.PLS.Pos4.Ok := FALSE;
   BookedExtractor.DrivePick.PLS.Pos5.LowLimit := 0.0;
   BookedExtractor.DrivePick.PLS.Pos5.HighLimit := 0.0;
   BookedExtractor.DrivePick.PLS.Pos5.Ok := FALSE;
   BookedExtractor.DrivePick.TON_EnableDrive.PT := T#500MS;
   BookedExtractor.DrivePick.TON_EnableDrive.IN := FALSE;
   BookedExtractor.DrivePick.TON_HwOvertravel_Dis.PT := T#0MS;
   BookedExtractor.DrivePick.TON_HwOvertravel_Dis.IN := FALSE;
   BookedExtractor.DrivePick.TON_HwOvertravel_En.PT := T#0MS;
   BookedExtractor.DrivePick.TON_HwOvertravel_En.IN := FALSE;
   BookedExtractor.DrivePick.TON_TimeoutMovement.PT := T#8S;
   BookedExtractor.DrivePick.TON_TimeoutMovement.IN := FALSE;
   BookedExtractor.DriveStore.AlmOk := FALSE;
   BookedExtractor.DriveStore.AlmEmerg := FALSE;
   BookedExtractor.DriveStore.AlmNode := FALSE;
   BookedExtractor.DriveStore.InitPosDrive := FALSE;
   BookedExtractor.DriveStore.InitPosDrivePLS := FALSE;
   BookedExtractor.DriveStore.GearingON := FALSE;
   BookedExtractor.DriveStore.CamHook := FALSE;
   BookedExtractor.DriveStore.CamStoppingPhase := FALSE;
   BookedExtractor.DriveStore.RepositioningRequest := FALSE;
   BookedExtractor.DriveStore.CamRequestResult := FALSE;
   BookedExtractor.DriveStore.CamRequestError := FALSE;
   BookedExtractor.DriveStore.CamRequestOk := FALSE;
   BookedExtractor.DriveStore.CalibDisAxisReq := FALSE;
   BookedExtractor.DriveStore.CalibReq := FALSE;
   BookedExtractor.DriveStore.CalibProcess := FALSE;
   BookedExtractor.DriveStore.HwOvertravelDisReq := FALSE;
   BookedExtractor.DriveStore.HwOvertravelEnReq := FALSE;
   BookedExtractor.DriveStore.AuxCamRequest := FALSE;
   BookedExtractor.DriveStore.TorquePeakEna := TRUE;
   BookedExtractor.DriveStore.Cmd_Repos := FALSE;
   BookedExtractor.DriveStore.Ons_CamRequest := FALSE;
   BookedExtractor.DriveStore.AuxCmdPosition := 0;
   BookedExtractor.DriveStore.Unwind := 80.0;
   BookedExtractor.DriveStore.MaxDev := 0.0;
   BookedExtractor.DriveStore.ReposSpeed := 100.0;
   BookedExtractor.DriveStore.CalcSlaveDifferenceABS := 0.0;
   BookedExtractor.DriveStore.CalcModPosition := 0.0;
   BookedExtractor.DriveStore.CalcSlaveDifference := 0.0;
   BookedExtractor.DriveStore.CalcMinDeltaPos := 0.0;
   BookedExtractor.DriveStore.CalcMaxDeltaPos := 0.0;
   BookedExtractor.DriveStore.CalcHalfPosUnwind := 0.0;
   BookedExtractor.DriveStore.Man.Cmd_PosJog := FALSE;
   BookedExtractor.DriveStore.Man.Cmd_NegJog := FALSE;
   BookedExtractor.DriveStore.Man.Cmd_Step := FALSE;
   BookedExtractor.DriveStore.Man.Cmd_Forward := FALSE;
   BookedExtractor.DriveStore.Man.Cmd_Backward := FALSE;
   BookedExtractor.DriveStore.Man.Cmd_Up := FALSE;
   BookedExtractor.DriveStore.Man.Cmd_Down := FALSE;
   BookedExtractor.DriveStore.Man.Cmd_Intermediate := FALSE;
   BookedExtractor.DriveStore.Man.Cmd_Open := FALSE;
   BookedExtractor.DriveStore.Man.Cmd_Close := FALSE;
   BookedExtractor.DriveStore.Man.Cmd_PreOpen := FALSE;
   BookedExtractor.DriveStore.Man.Cmd_Maintenance := FALSE;
   BookedExtractor.DriveStore.Man.Cmd_OperatorSide := FALSE;
   BookedExtractor.DriveStore.Man.Cmd_NotOperatorSide := FALSE;
   BookedExtractor.DriveStore.Man.Cmd_OnMould := FALSE;
   BookedExtractor.DriveStore.Man.Cmd_OffMould := FALSE;
   BookedExtractor.DriveStore.Man.Cmd_Pos0 := FALSE;
   BookedExtractor.DriveStore.Man.Cmd_Pos1 := FALSE;
   BookedExtractor.DriveStore.Man.Cmd_Pos2 := FALSE;
   BookedExtractor.DriveStore.Man.Cmd_Pos3 := FALSE;
   BookedExtractor.DriveStore.Man.Cmd_Pos4 := FALSE;
   BookedExtractor.DriveStore.Man.Cmd_Pos5 := FALSE;
   BookedExtractor.DriveStore.Man.Ons_Step := FALSE;
   BookedExtractor.DriveStore.Man.PhaseJogCmd := FALSE;
   BookedExtractor.DriveStore.Man.CmdStartStep := FALSE;
   BookedExtractor.DriveStore.Man.CmdEndStep := FALSE;
   BookedExtractor.DriveStore.Man.StepCond := FALSE;
   BookedExtractor.DriveStore.Man.TON_DelayHomeCmd.PT := T#3S;
   BookedExtractor.DriveStore.Man.TON_DelayHomeCmd.IN := FALSE;
   BookedExtractor.DriveStore.Auto.Cmd_Step := FALSE;
   BookedExtractor.DriveStore.Auto.Cmd_StartStep := FALSE;
   BookedExtractor.DriveStore.Auto.Cmd_EndStep := FALSE;
   BookedExtractor.DriveStore.Auto.Cmd_Forward := FALSE;
   BookedExtractor.DriveStore.Auto.Cmd_Backward := FALSE;
   BookedExtractor.DriveStore.Auto.Cmd_Up := FALSE;
   BookedExtractor.DriveStore.Auto.Cmd_Down := FALSE;
   BookedExtractor.DriveStore.Auto.Cmd_Intermediate := FALSE;
   BookedExtractor.DriveStore.Auto.Cmd_Open := FALSE;
   BookedExtractor.DriveStore.Auto.Cmd_Close := FALSE;
   BookedExtractor.DriveStore.Auto.Cmd_PreOpen := FALSE;
   BookedExtractor.DriveStore.Auto.Cmd_Maintenance := FALSE;
   BookedExtractor.DriveStore.Auto.Cmd_OperatorSide := FALSE;
   BookedExtractor.DriveStore.Auto.Cmd_NotOperatorSide := FALSE;
   BookedExtractor.DriveStore.Auto.Cmd_OnMould := FALSE;
   BookedExtractor.DriveStore.Auto.Cmd_OffMould := FALSE;
   BookedExtractor.DriveStore.Auto.Cmd_Pos0 := FALSE;
   BookedExtractor.DriveStore.Auto.Cmd_Pos1 := FALSE;
   BookedExtractor.DriveStore.Auto.Cmd_Pos2 := FALSE;
   BookedExtractor.DriveStore.Auto.Cmd_Pos3 := FALSE;
   BookedExtractor.DriveStore.Auto.Cmd_Pos4 := FALSE;
   BookedExtractor.DriveStore.Auto.Cmd_Pos5 := FALSE;
   BookedExtractor.DriveStore.Auto.Cmd_Gear := FALSE;
   BookedExtractor.DriveStore.ACT.CMD.Enable := FALSE;
   BookedExtractor.DriveStore.ACT.CMD.Pos_Mode := FALSE;
   BookedExtractor.DriveStore.ACT.CMD.MergeDisabled := FALSE;
   BookedExtractor.DriveStore.ACT.CMD.SCurve := FALSE;
   BookedExtractor.DriveStore.ACT.CMD.Cam_Mode := FALSE;
   BookedExtractor.DriveStore.ACT.CMD.Cam_Request := FALSE;
   BookedExtractor.DriveStore.ACT.CMD.Cam_PhaseStop := FALSE;
   BookedExtractor.DriveStore.ACT.CMD.Gear_Mode := FALSE;
   BookedExtractor.DriveStore.ACT.CMD.Repos_Req := FALSE;
   BookedExtractor.DriveStore.ACT.CMD.Jog_Pos := FALSE;
   BookedExtractor.DriveStore.ACT.CMD.Jog_Neg := FALSE;
   BookedExtractor.DriveStore.ACT.CMD.Stop := TRUE;
   BookedExtractor.DriveStore.ACT.CMD.Calibration_Req := FALSE;
   BookedExtractor.DriveStore.ACT.CMD.Reset := FALSE;
   BookedExtractor.DriveStore.ACT.CMD.RegInput1 := FALSE;
   BookedExtractor.DriveStore.ACT.CMD.Brake_Release := FALSE;
   BookedExtractor.DriveStore.ACT.CMD.HwPosOvertravel_Dis := FALSE;
   BookedExtractor.DriveStore.ACT.CMD.HwNegOvertravel_Dis := FALSE;
   BookedExtractor.DriveStore.ACT.CMD.HwOvertravel_MSG_En := FALSE;
   BookedExtractor.DriveStore.ACT.CMD.OneShootMove := FALSE;
   BookedExtractor.DriveStore.ACT.CMD.Move_Type := 3;
   BookedExtractor.DriveStore.ACT.CMD.Target_Pos := 0.0;
   BookedExtractor.DriveStore.ACT.CMD.Speed := 100.0;
   BookedExtractor.DriveStore.ACT.CMD.Acceleration := 100.0;
   BookedExtractor.DriveStore.ACT.CMD.Deceleration := 4500.0;
   BookedExtractor.DriveStore.ACT.CMD.Torque_Limit := 15.0;
   BookedExtractor.DriveStore.ACT.CMD.Gear_Ratio := 0.0;
   BookedExtractor.DriveStore.ACT.CMD.Mccp_Length := 0;
   BookedExtractor.DriveStore.ACT.CMD.Mccp_StartSlope := 0.0;
   BookedExtractor.DriveStore.ACT.CMD.Mccp_EndSlope := 0.0;
   BookedExtractor.DriveStore.ACT.CMD.Mapc_Direction := 0;
   BookedExtractor.DriveStore.ACT.CMD.Mapc_SlaveScaling := 0.0;
   BookedExtractor.DriveStore.ACT.CMD.Mapc_MasterScaling := 0.0;
   BookedExtractor.DriveStore.ACT.CMD.Mapc_MasterLockPosition := 0.0;
   BookedExtractor.DriveStore.ACT.CMD.Mapc_CamLockPosition := 0.0;
   BookedExtractor.DriveStore.ACT.CMD.Cam[0..39].leadingValueStart := 0.0;
   BookedExtractor.DriveStore.ACT.CMD.Cam[0..39].leadingValueEnd := 0.0;
   BookedExtractor.DriveStore.ACT.CMD.Cam[0..39].followingValueStart := 0.0;
   BookedExtractor.DriveStore.ACT.CMD.Cam[0..39].followingValueEnd := 0.0;
   BookedExtractor.DriveStore.ACT.CMD.Cam[0..39].geoVeloStart := 0.0;
   BookedExtractor.DriveStore.ACT.CMD.Cam[0..39].geoVeloEnd := 0.0;
   BookedExtractor.DriveStore.ACT.CMD.Cam[0..39].geoAccelStart := 0.0;
   BookedExtractor.DriveStore.ACT.CMD.Cam[0..39].geoAccelEnd := 0.0;
   BookedExtractor.DriveStore.ACT.CMD.Cam[0..39].geoJerkStart := 0.0;
   BookedExtractor.DriveStore.ACT.CMD.Cam[0..39].geoJerkEnd := 0.0;
   BookedExtractor.DriveStore.ACT.CMD.Cam[0..39].inflectionPointParameter := 0.5;
   BookedExtractor.DriveStore.ACT.CMD.Cam[0..39].modVeloTrapezoidParameter := 1.0;
   BookedExtractor.DriveStore.ACT.CMD.Cam[0..39].modSineMaxAccelCaStar := 0.0;
   BookedExtractor.DriveStore.ACT.CMD.Cam[0..39].camProfileType := 0;
   BookedExtractor.DriveStore.ACT.FBK.Ready := TRUE;
   BookedExtractor.DriveStore.ACT.FBK.Calibrated := TRUE;
   BookedExtractor.DriveStore.ACT.FBK.Fault := FALSE;
   BookedExtractor.DriveStore.ACT.FBK.ModuleConnFault := FALSE;
   BookedExtractor.DriveStore.ACT.FBK.In_Position := FALSE;
   BookedExtractor.DriveStore.ACT.FBK.Standstill := TRUE;
   BookedExtractor.DriveStore.ACT.FBK.Enabled := FALSE;
   BookedExtractor.DriveStore.ACT.FBK.BusReadyStatus := FALSE;
   BookedExtractor.DriveStore.ACT.FBK.BrakeReleased := FALSE;
   BookedExtractor.DriveStore.ACT.FBK.HwPosOvertravelDisabled := FALSE;
   BookedExtractor.DriveStore.ACT.FBK.HwNegOvertravelDisabled := FALSE;
   BookedExtractor.DriveStore.ACT.FBK.SafeOffStatus := FALSE;
   BookedExtractor.DriveStore.ACT.FBK.MaxTorqueLimit := FALSE;
   BookedExtractor.DriveStore.ACT.FBK.PosMerge_IP := FALSE;
   BookedExtractor.DriveStore.ACT.FBK.PosMerge_PC := FALSE;
   BookedExtractor.DriveStore.ACT.FBK.Gearing_IP := FALSE;
   BookedExtractor.DriveStore.ACT.FBK.Position := 0.0;
   BookedExtractor.DriveStore.ACT.FBK.Speed := 0.0;
   BookedExtractor.DriveStore.ACT.FBK.Torque := 0.0;
   BookedExtractor.DriveStore.ACT.FBK.RegInput1Pos := 0.0;
   BookedExtractor.DriveStore.ACT.FBK.SeqCamErrorCode := 0;
   BookedExtractor.DriveStore.ACT.FBK.SeqCamTargetPosMAM := 0.0;
   BookedExtractor.DriveStore.ACT.FBK.SeqCamStatus.EndSequence := FALSE;
   BookedExtractor.DriveStore.ACT.FBK.SeqCamStatus.EndSuccess := FALSE;
   BookedExtractor.DriveStore.ACT.FBK.SeqCamStatus.EndError := FALSE;
   BookedExtractor.DriveStore.ACT.FBK.SeqCamStatus.CamHook := FALSE;
   BookedExtractor.DriveStore.ACT.FBK.SeqCamStatus.BothMapc_IP := FALSE;
   BookedExtractor.DriveStore.ACT.FBK.SeqCamStatus.SlaveFwd := FALSE;
   BookedExtractor.DriveStore.ACT.FBK.SeqCamStatus.SlaveBwd := FALSE;
   BookedExtractor.DriveStore.ACT.FBK.SeqCamStatus.SlaveUnwind := FALSE;
   BookedExtractor.DriveStore.ACT.FBK.SeqCamStatus.WaitValidByOpe := FALSE;
   BookedExtractor.DriveStore.ACT.FBK.SeqCamStatus.MapcA_IP := FALSE;
   BookedExtractor.DriveStore.ACT.FBK.SeqCamStatus.MapcB_IP := FALSE;
   BookedExtractor.DriveStore.ACT.FBK.SeqCamStatus.MapcC_IP := FALSE;
   BookedExtractor.DriveStore.ACT.FBK.SeqCamStatus.CamOnce_PC := FALSE;
   BookedExtractor.DriveStore.ACT.FBK.SeqCamStatus.MaxDevError := FALSE;
   BookedExtractor.DriveStore.ACT.FBK.SeqCamStatus.PositionCamLockStatus := FALSE;
   BookedExtractor.DriveStore.ACT.FBK.SeqCamStatus.WaitRestart := FALSE;
   BookedExtractor.DriveStore.ACT.FBK.SeqCamStatus.Bit17 := FALSE;
   BookedExtractor.DriveStore.ACT.FBK.SeqCamStatus.Bit18 := FALSE;
   BookedExtractor.DriveStore.ACT.FBK.SeqCamStatus.Bit19 := FALSE;
   BookedExtractor.DriveStore.ACT.FBK.SeqCamStatus.Bit20 := FALSE;
   BookedExtractor.DriveStore.ACT.FBK.SeqCamStatus.Bit21 := FALSE;
   BookedExtractor.DriveStore.ACT.FBK.SeqCamStatus.Bit22 := FALSE;
   BookedExtractor.DriveStore.ACT.FBK.SeqCamStatus.Bit23 := FALSE;
   BookedExtractor.DriveStore.ACT.FBK.SeqCamStatus.Bit24 := FALSE;
   BookedExtractor.DriveStore.ACT.FBK.SeqCamStatus.Bit25 := FALSE;
   BookedExtractor.DriveStore.ACT.FBK.SeqCamStatus.Bit26 := FALSE;
   BookedExtractor.DriveStore.ACT.FBK.SeqCamStatus.Bit27 := FALSE;
   BookedExtractor.DriveStore.ACT.FBK.SeqCamStatus.Bit28 := FALSE;
   BookedExtractor.DriveStore.ACT.FBK.SeqCamStatus.Bit29 := FALSE;
   BookedExtractor.DriveStore.ACT.FBK.SeqCamStatus.Bit30 := FALSE;
   BookedExtractor.DriveStore.ACT.FBK.SeqCamStatus.Bit31 := FALSE;
   BookedExtractor.DriveStore.ACT.FBK.SeqCamStatus.Bit32 := FALSE;
   BookedExtractor.DriveStore.PLS.FinePosOk.LowLimit := 79.0;
   BookedExtractor.DriveStore.PLS.FinePosOk.HighLimit := 1.0;
   BookedExtractor.DriveStore.PLS.FinePosOk.Ok := TRUE;
   BookedExtractor.DriveStore.PLS.KeepPosOk.LowLimit := 0.0;
   BookedExtractor.DriveStore.PLS.KeepPosOk.HighLimit := 0.0;
   BookedExtractor.DriveStore.PLS.KeepPosOk.Ok := FALSE;
   BookedExtractor.DriveStore.PLS.Up.LowLimit := 0.0;
   BookedExtractor.DriveStore.PLS.Up.HighLimit := 0.0;
   BookedExtractor.DriveStore.PLS.Up.Ok := FALSE;
   BookedExtractor.DriveStore.PLS.Intermediate.LowLimit := 0.0;
   BookedExtractor.DriveStore.PLS.Intermediate.HighLimit := 0.0;
   BookedExtractor.DriveStore.PLS.Intermediate.Ok := FALSE;
   BookedExtractor.DriveStore.PLS.Down.LowLimit := 0.0;
   BookedExtractor.DriveStore.PLS.Down.HighLimit := 0.0;
   BookedExtractor.DriveStore.PLS.Down.Ok := FALSE;
   BookedExtractor.DriveStore.PLS.Forward.LowLimit := 0.0;
   BookedExtractor.DriveStore.PLS.Forward.HighLimit := 0.0;
   BookedExtractor.DriveStore.PLS.Forward.Ok := FALSE;
   BookedExtractor.DriveStore.PLS.Backward.LowLimit := 0.0;
   BookedExtractor.DriveStore.PLS.Backward.HighLimit := 0.0;
   BookedExtractor.DriveStore.PLS.Backward.Ok := FALSE;
   BookedExtractor.DriveStore.PLS.Open.LowLimit := 0.0;
   BookedExtractor.DriveStore.PLS.Open.HighLimit := 0.0;
   BookedExtractor.DriveStore.PLS.Open.Ok := FALSE;
   BookedExtractor.DriveStore.PLS.Close.LowLimit := 0.0;
   BookedExtractor.DriveStore.PLS.Close.HighLimit := 0.0;
   BookedExtractor.DriveStore.PLS.Close.Ok := FALSE;
   BookedExtractor.DriveStore.PLS.PreOpen.LowLimit := 0.0;
   BookedExtractor.DriveStore.PLS.PreOpen.HighLimit := 0.0;
   BookedExtractor.DriveStore.PLS.PreOpen.Ok := FALSE;
   BookedExtractor.DriveStore.PLS.Maintenance.LowLimit := 0.0;
   BookedExtractor.DriveStore.PLS.Maintenance.HighLimit := 0.0;
   BookedExtractor.DriveStore.PLS.Maintenance.Ok := FALSE;
   BookedExtractor.DriveStore.PLS.OperatorSide.LowLimit := 0.0;
   BookedExtractor.DriveStore.PLS.OperatorSide.HighLimit := 0.0;
   BookedExtractor.DriveStore.PLS.OperatorSide.Ok := FALSE;
   BookedExtractor.DriveStore.PLS.NotOperatorSide.LowLimit := 0.0;
   BookedExtractor.DriveStore.PLS.NotOperatorSide.HighLimit := 0.0;
   BookedExtractor.DriveStore.PLS.NotOperatorSide.Ok := FALSE;
   BookedExtractor.DriveStore.PLS.OnMould.LowLimit := 0.0;
   BookedExtractor.DriveStore.PLS.OnMould.HighLimit := 0.0;
   BookedExtractor.DriveStore.PLS.OnMould.Ok := FALSE;
   BookedExtractor.DriveStore.PLS.OffMould.LowLimit := 0.0;
   BookedExtractor.DriveStore.PLS.OffMould.HighLimit := 0.0;
   BookedExtractor.DriveStore.PLS.OffMould.Ok := FALSE;
   BookedExtractor.DriveStore.PLS.Pos0.LowLimit := 0.0;
   BookedExtractor.DriveStore.PLS.Pos0.HighLimit := 0.0;
   BookedExtractor.DriveStore.PLS.Pos0.Ok := FALSE;
   BookedExtractor.DriveStore.PLS.Pos1.LowLimit := 0.0;
   BookedExtractor.DriveStore.PLS.Pos1.HighLimit := 0.0;
   BookedExtractor.DriveStore.PLS.Pos1.Ok := FALSE;
   BookedExtractor.DriveStore.PLS.Pos2.LowLimit := 0.0;
   BookedExtractor.DriveStore.PLS.Pos2.HighLimit := 0.0;
   BookedExtractor.DriveStore.PLS.Pos2.Ok := FALSE;
   BookedExtractor.DriveStore.PLS.Pos3.LowLimit := 0.0;
   BookedExtractor.DriveStore.PLS.Pos3.HighLimit := 0.0;
   BookedExtractor.DriveStore.PLS.Pos3.Ok := FALSE;
   BookedExtractor.DriveStore.PLS.Pos4.LowLimit := 0.0;
   BookedExtractor.DriveStore.PLS.Pos4.HighLimit := 0.0;
   BookedExtractor.DriveStore.PLS.Pos4.Ok := FALSE;
   BookedExtractor.DriveStore.PLS.Pos5.LowLimit := 0.0;
   BookedExtractor.DriveStore.PLS.Pos5.HighLimit := 0.0;
   BookedExtractor.DriveStore.PLS.Pos5.Ok := FALSE;
   BookedExtractor.DriveStore.TON_EnableDrive.PT := T#500MS;
   BookedExtractor.DriveStore.TON_EnableDrive.IN := FALSE;
   BookedExtractor.DriveStore.TON_HwOvertravel_Dis.PT := T#0MS;
   BookedExtractor.DriveStore.TON_HwOvertravel_Dis.IN := FALSE;
   BookedExtractor.DriveStore.TON_HwOvertravel_En.PT := T#0MS;
   BookedExtractor.DriveStore.TON_HwOvertravel_En.IN := FALSE;
   BookedExtractor.DriveStore.TON_TimeoutMovement.PT := T#8S;
   BookedExtractor.DriveStore.TON_TimeoutMovement.IN := FALSE;
   BookedExtractor.TON_ResetMaxLevel.PT := T#2S;
   BookedExtractor.TON_ResetMaxLevel.ET := T#2S;
   BookedExtractor.TON_ResetMaxLevel.IN := TRUE;
   BookedExtractor.TON_ResetMaxLevel.Q := TRUE;
   BookedExtractor.RTO_Work.PT := T#1M;
   BookedExtractor.RTO_Work.IN := FALSE;
   BookedExtractor.TON_ScOK.PT := T#20S;
   BookedExtractor.TON_ScOK.IN := FALSE;
   BookedExtractor.TON_IncorrectPosOpeSide.PT := T#4S;
   BookedExtractor.TON_IncorrectPosOpeSide.IN := FALSE;
   BookedExtractor.TON_IncorrectPosNotOpeSide.PT := T#4S;
   BookedExtractor.TON_IncorrectPosNotOpeSide.IN := FALSE;
   BookedExtractor.TON_Sign_MaxLevel.PT := T#1S;
   BookedExtractor.TON_Sign_MaxLevel.IN := FALSE;
   BookedExtractor.TON_TimeoutWork.PT := T#20S;
   BookedExtractor.TON_TimeoutWork.IN := FALSE;
   DropInserter.ScOk := FALSE;
   DropInserter.CycleOn := FALSE;
   DropInserter.Work := FALSE;
   DropInserter.OkToStop := FALSE;
   DropInserter.AlmOk := TRUE;
   DropInserter.DrivesEnabled := FALSE;
   DropInserter.OutChainObstruction := FALSE;
   DropInserter.SingleCycle := FALSE;
   DropInserter.RepositioningReq := FALSE;
   DropInserter.Ons_TimeWork := FALSE;
   DropInserter.NumMinLevel := 0;
   DropInserter.Input.MouPreIns := FALSE;
   DropInserter.Input.EnaSel := FALSE;
   DropInserter.Input.MinLvl := FALSE;
   DropInserter.Input.TabOn := FALSE;
   DropInserter.Input.TabOff := FALSE;
   DropInserter.Output.EnaSelLgh := FALSE;
   DropInserter.Output.TabOn := FALSE;
   DropInserter.Output.TabOff := FALSE;
   DropInserter.Man.Ons_SingleCycle := FALSE;
   DropInserter.Man.CmdTurntableStraight := FALSE;
   DropInserter.Man.CmdTurntableTilted := FALSE;
   DropInserter.Man.CmdSingleCycle := FALSE;
   DropInserter.Man.EnaPbt := FALSE;
   DropInserter.Man.RstCmd := FALSE;
   DropInserter.Man.ScreenNumber := 302_070_301;
   DropInserter.Man.WithinScreenRange := 0;
   DropInserter."Step"._00_CycleActivated_OpenStorageCmd := FALSE;
   DropInserter."Step"._10_OpenStoragePos := FALSE;
   DropInserter."Step"._20_CloseStorageCmd := FALSE;
   DropInserter."Step"._30_CloseStoragePos_TableStraightCmd := FALSE;
   DropInserter."Step"._40_TableStraightPos_PreOpenStorageCmd := FALSE;
   DropInserter."Step"._50_PreOpenStoragePos_TableTiltedCmd := FALSE;
   DropInserter."Step"._60_TableTiltedPos_EndCycle := FALSE;
   DropInserter."Step".ons_StrobeWorkDone := FALSE;
   DropInserter."Step".StrobeWorkDone := FALSE;
   DropInserter."Step".ScSeqOk := FALSE;
   DropInserter."Step".SeqActive := FALSE;
   DropInserter.Drive.AlmOk := FALSE;
   DropInserter.Drive.AlmEmerg := FALSE;
   DropInserter.Drive.AlmNode := FALSE;
   DropInserter.Drive.InitPosDrive := FALSE;
   DropInserter.Drive.InitPosDrivePLS := FALSE;
   DropInserter.Drive.GearingON := FALSE;
   DropInserter.Drive.CamHook := FALSE;
   DropInserter.Drive.CamStoppingPhase := FALSE;
   DropInserter.Drive.RepositioningRequest := FALSE;
   DropInserter.Drive.CamRequestResult := FALSE;
   DropInserter.Drive.CamRequestError := FALSE;
   DropInserter.Drive.CamRequestOk := FALSE;
   DropInserter.Drive.CalibDisAxisReq := FALSE;
   DropInserter.Drive.CalibReq := FALSE;
   DropInserter.Drive.CalibProcess := FALSE;
   DropInserter.Drive.HwOvertravelDisReq := FALSE;
   DropInserter.Drive.HwOvertravelEnReq := FALSE;
   DropInserter.Drive.AuxCamRequest := FALSE;
   DropInserter.Drive.TorquePeakEna := FALSE;
   DropInserter.Drive.Cmd_Repos := FALSE;
   DropInserter.Drive.Ons_CamRequest := FALSE;
   DropInserter.Drive.AuxCmdPosition := 0;
   DropInserter.Drive.Unwind := 0.0;
   DropInserter.Drive.MaxDev := 0.0;
   DropInserter.Drive.ReposSpeed := 100.0;
   DropInserter.Drive.CalcSlaveDifferenceABS := 0.0;
   DropInserter.Drive.CalcModPosition := 0.0;
   DropInserter.Drive.CalcSlaveDifference := 0.0;
   DropInserter.Drive.CalcMinDeltaPos := 0.0;
   DropInserter.Drive.CalcMaxDeltaPos := 0.0;
   DropInserter.Drive.CalcHalfPosUnwind := 0.0;
   DropInserter.Drive.Man.Cmd_PosJog := FALSE;
   DropInserter.Drive.Man.Cmd_NegJog := FALSE;
   DropInserter.Drive.Man.Cmd_Step := FALSE;
   DropInserter.Drive.Man.Cmd_Forward := FALSE;
   DropInserter.Drive.Man.Cmd_Backward := FALSE;
   DropInserter.Drive.Man.Cmd_Up := FALSE;
   DropInserter.Drive.Man.Cmd_Down := FALSE;
   DropInserter.Drive.Man.Cmd_Intermediate := FALSE;
   DropInserter.Drive.Man.Cmd_Open := FALSE;
   DropInserter.Drive.Man.Cmd_Close := FALSE;
   DropInserter.Drive.Man.Cmd_PreOpen := FALSE;
   DropInserter.Drive.Man.Cmd_Maintenance := FALSE;
   DropInserter.Drive.Man.Cmd_OperatorSide := FALSE;
   DropInserter.Drive.Man.Cmd_NotOperatorSide := FALSE;
   DropInserter.Drive.Man.Cmd_OnMould := FALSE;
   DropInserter.Drive.Man.Cmd_OffMould := FALSE;
   DropInserter.Drive.Man.Cmd_Pos0 := FALSE;
   DropInserter.Drive.Man.Cmd_Pos1 := FALSE;
   DropInserter.Drive.Man.Cmd_Pos2 := FALSE;
   DropInserter.Drive.Man.Cmd_Pos3 := FALSE;
   DropInserter.Drive.Man.Cmd_Pos4 := FALSE;
   DropInserter.Drive.Man.Cmd_Pos5 := FALSE;
   DropInserter.Drive.Man.Ons_Step := FALSE;
   DropInserter.Drive.Man.PhaseJogCmd := FALSE;
   DropInserter.Drive.Man.CmdStartStep := FALSE;
   DropInserter.Drive.Man.CmdEndStep := FALSE;
   DropInserter.Drive.Man.StepCond := FALSE;
   DropInserter.Drive.Man.TON_DelayHomeCmd.PT := T#3S;
   DropInserter.Drive.Man.TON_DelayHomeCmd.IN := FALSE;
   DropInserter.Drive.Auto.Cmd_Step := FALSE;
   DropInserter.Drive.Auto.Cmd_StartStep := FALSE;
   DropInserter.Drive.Auto.Cmd_EndStep := FALSE;
   DropInserter.Drive.Auto.Cmd_Forward := FALSE;
   DropInserter.Drive.Auto.Cmd_Backward := FALSE;
   DropInserter.Drive.Auto.Cmd_Up := FALSE;
   DropInserter.Drive.Auto.Cmd_Down := FALSE;
   DropInserter.Drive.Auto.Cmd_Intermediate := FALSE;
   DropInserter.Drive.Auto.Cmd_Open := FALSE;
   DropInserter.Drive.Auto.Cmd_Close := FALSE;
   DropInserter.Drive.Auto.Cmd_PreOpen := FALSE;
   DropInserter.Drive.Auto.Cmd_Maintenance := FALSE;
   DropInserter.Drive.Auto.Cmd_OperatorSide := FALSE;
   DropInserter.Drive.Auto.Cmd_NotOperatorSide := FALSE;
   DropInserter.Drive.Auto.Cmd_OnMould := FALSE;
   DropInserter.Drive.Auto.Cmd_OffMould := FALSE;
   DropInserter.Drive.Auto.Cmd_Pos0 := FALSE;
   DropInserter.Drive.Auto.Cmd_Pos1 := FALSE;
   DropInserter.Drive.Auto.Cmd_Pos2 := FALSE;
   DropInserter.Drive.Auto.Cmd_Pos3 := FALSE;
   DropInserter.Drive.Auto.Cmd_Pos4 := FALSE;
   DropInserter.Drive.Auto.Cmd_Pos5 := FALSE;
   DropInserter.Drive.Auto.Cmd_Gear := FALSE;
   DropInserter.Drive.ACT.CMD.Enable := FALSE;
   DropInserter.Drive.ACT.CMD.Pos_Mode := FALSE;
   DropInserter.Drive.ACT.CMD.MergeDisabled := FALSE;
   DropInserter.Drive.ACT.CMD.SCurve := FALSE;
   DropInserter.Drive.ACT.CMD.Cam_Mode := FALSE;
   DropInserter.Drive.ACT.CMD.Cam_Request := FALSE;
   DropInserter.Drive.ACT.CMD.Cam_PhaseStop := FALSE;
   DropInserter.Drive.ACT.CMD.Gear_Mode := FALSE;
   DropInserter.Drive.ACT.CMD.Repos_Req := FALSE;
   DropInserter.Drive.ACT.CMD.Jog_Pos := FALSE;
   DropInserter.Drive.ACT.CMD.Jog_Neg := FALSE;
   DropInserter.Drive.ACT.CMD.Stop := FALSE;
   DropInserter.Drive.ACT.CMD.Calibration_Req := FALSE;
   DropInserter.Drive.ACT.CMD.Reset := FALSE;
   DropInserter.Drive.ACT.CMD.RegInput1 := FALSE;
   DropInserter.Drive.ACT.CMD.Brake_Release := FALSE;
   DropInserter.Drive.ACT.CMD.HwPosOvertravel_Dis := FALSE;
   DropInserter.Drive.ACT.CMD.HwNegOvertravel_Dis := FALSE;
   DropInserter.Drive.ACT.CMD.HwOvertravel_MSG_En := FALSE;
   DropInserter.Drive.ACT.CMD.OneShootMove := FALSE;
   DropInserter.Drive.ACT.CMD.Move_Type := 0;
   DropInserter.Drive.ACT.CMD.Target_Pos := 0.0;
   DropInserter.Drive.ACT.CMD.Speed := 0.0;
   DropInserter.Drive.ACT.CMD.Acceleration := 0.0;
   DropInserter.Drive.ACT.CMD.Deceleration := 0.0;
   DropInserter.Drive.ACT.CMD.Torque_Limit := 0.0;
   DropInserter.Drive.ACT.CMD.Gear_Ratio := 0.0;
   DropInserter.Drive.ACT.CMD.Mccp_Length := 0;
   DropInserter.Drive.ACT.CMD.Mccp_StartSlope := 0.0;
   DropInserter.Drive.ACT.CMD.Mccp_EndSlope := 0.0;
   DropInserter.Drive.ACT.CMD.Mapc_Direction := 0;
   DropInserter.Drive.ACT.CMD.Mapc_SlaveScaling := 0.0;
   DropInserter.Drive.ACT.CMD.Mapc_MasterScaling := 0.0;
   DropInserter.Drive.ACT.CMD.Mapc_MasterLockPosition := 0.0;
   DropInserter.Drive.ACT.CMD.Mapc_CamLockPosition := 0.0;
   DropInserter.Drive.ACT.CMD.Cam[0..39].leadingValueStart := 0.0;
   DropInserter.Drive.ACT.CMD.Cam[0..39].leadingValueEnd := 0.0;
   DropInserter.Drive.ACT.CMD.Cam[0..39].followingValueStart := 0.0;
   DropInserter.Drive.ACT.CMD.Cam[0..39].followingValueEnd := 0.0;
   DropInserter.Drive.ACT.CMD.Cam[0..39].geoVeloStart := 0.0;
   DropInserter.Drive.ACT.CMD.Cam[0..39].geoVeloEnd := 0.0;
   DropInserter.Drive.ACT.CMD.Cam[0..39].geoAccelStart := 0.0;
   DropInserter.Drive.ACT.CMD.Cam[0..39].geoAccelEnd := 0.0;
   DropInserter.Drive.ACT.CMD.Cam[0..39].geoJerkStart := 0.0;
   DropInserter.Drive.ACT.CMD.Cam[0..39].geoJerkEnd := 0.0;
   DropInserter.Drive.ACT.CMD.Cam[0..39].inflectionPointParameter := 0.5;
   DropInserter.Drive.ACT.CMD.Cam[0..39].modVeloTrapezoidParameter := 1.0;
   DropInserter.Drive.ACT.CMD.Cam[0..39].modSineMaxAccelCaStar := 0.0;
   DropInserter.Drive.ACT.CMD.Cam[0..39].camProfileType := 0;
   DropInserter.Drive.ACT.FBK.Ready := FALSE;
   DropInserter.Drive.ACT.FBK.Calibrated := FALSE;
   DropInserter.Drive.ACT.FBK.Fault := FALSE;
   DropInserter.Drive.ACT.FBK.ModuleConnFault := FALSE;
   DropInserter.Drive.ACT.FBK.In_Position := FALSE;
   DropInserter.Drive.ACT.FBK.Standstill := FALSE;
   DropInserter.Drive.ACT.FBK.Enabled := FALSE;
   DropInserter.Drive.ACT.FBK.BusReadyStatus := FALSE;
   DropInserter.Drive.ACT.FBK.BrakeReleased := FALSE;
   DropInserter.Drive.ACT.FBK.HwPosOvertravelDisabled := FALSE;
   DropInserter.Drive.ACT.FBK.HwNegOvertravelDisabled := FALSE;
   DropInserter.Drive.ACT.FBK.SafeOffStatus := FALSE;
   DropInserter.Drive.ACT.FBK.MaxTorqueLimit := FALSE;
   DropInserter.Drive.ACT.FBK.PosMerge_IP := FALSE;
   DropInserter.Drive.ACT.FBK.PosMerge_PC := FALSE;
   DropInserter.Drive.ACT.FBK.Gearing_IP := FALSE;
   DropInserter.Drive.ACT.FBK.Position := 0.0;
   DropInserter.Drive.ACT.FBK.Speed := 0.0;
   DropInserter.Drive.ACT.FBK.Torque := 0.0;
   DropInserter.Drive.ACT.FBK.RegInput1Pos := 0.0;
   DropInserter.Drive.ACT.FBK.SeqCamErrorCode := 0;
   DropInserter.Drive.ACT.FBK.SeqCamTargetPosMAM := 0.0;
   DropInserter.Drive.ACT.FBK.SeqCamStatus.EndSequence := FALSE;
   DropInserter.Drive.ACT.FBK.SeqCamStatus.EndSuccess := FALSE;
   DropInserter.Drive.ACT.FBK.SeqCamStatus.EndError := FALSE;
   DropInserter.Drive.ACT.FBK.SeqCamStatus.CamHook := FALSE;
   DropInserter.Drive.ACT.FBK.SeqCamStatus.BothMapc_IP := FALSE;
   DropInserter.Drive.ACT.FBK.SeqCamStatus.SlaveFwd := FALSE;
   DropInserter.Drive.ACT.FBK.SeqCamStatus.SlaveBwd := FALSE;
   DropInserter.Drive.ACT.FBK.SeqCamStatus.SlaveUnwind := FALSE;
   DropInserter.Drive.ACT.FBK.SeqCamStatus.WaitValidByOpe := FALSE;
   DropInserter.Drive.ACT.FBK.SeqCamStatus.MapcA_IP := FALSE;
   DropInserter.Drive.ACT.FBK.SeqCamStatus.MapcB_IP := FALSE;
   DropInserter.Drive.ACT.FBK.SeqCamStatus.MapcC_IP := FALSE;
   DropInserter.Drive.ACT.FBK.SeqCamStatus.CamOnce_PC := FALSE;
   DropInserter.Drive.ACT.FBK.SeqCamStatus.MaxDevError := FALSE;
   DropInserter.Drive.ACT.FBK.SeqCamStatus.PositionCamLockStatus := FALSE;
   DropInserter.Drive.ACT.FBK.SeqCamStatus.WaitRestart := FALSE;
   DropInserter.Drive.ACT.FBK.SeqCamStatus.Bit17 := FALSE;
   DropInserter.Drive.ACT.FBK.SeqCamStatus.Bit18 := FALSE;
   DropInserter.Drive.ACT.FBK.SeqCamStatus.Bit19 := FALSE;
   DropInserter.Drive.ACT.FBK.SeqCamStatus.Bit20 := FALSE;
   DropInserter.Drive.ACT.FBK.SeqCamStatus.Bit21 := FALSE;
   DropInserter.Drive.ACT.FBK.SeqCamStatus.Bit22 := FALSE;
   DropInserter.Drive.ACT.FBK.SeqCamStatus.Bit23 := FALSE;
   DropInserter.Drive.ACT.FBK.SeqCamStatus.Bit24 := FALSE;
   DropInserter.Drive.ACT.FBK.SeqCamStatus.Bit25 := FALSE;
   DropInserter.Drive.ACT.FBK.SeqCamStatus.Bit26 := FALSE;
   DropInserter.Drive.ACT.FBK.SeqCamStatus.Bit27 := FALSE;
   DropInserter.Drive.ACT.FBK.SeqCamStatus.Bit28 := FALSE;
   DropInserter.Drive.ACT.FBK.SeqCamStatus.Bit29 := FALSE;
   DropInserter.Drive.ACT.FBK.SeqCamStatus.Bit30 := FALSE;
   DropInserter.Drive.ACT.FBK.SeqCamStatus.Bit31 := FALSE;
   DropInserter.Drive.ACT.FBK.SeqCamStatus.Bit32 := FALSE;
   DropInserter.Drive.PLS.FinePosOk.LowLimit := 0.0;
   DropInserter.Drive.PLS.FinePosOk.HighLimit := 0.0;
   DropInserter.Drive.PLS.FinePosOk.Ok := FALSE;
   DropInserter.Drive.PLS.KeepPosOk.LowLimit := 0.0;
   DropInserter.Drive.PLS.KeepPosOk.HighLimit := 0.0;
   DropInserter.Drive.PLS.KeepPosOk.Ok := FALSE;
   DropInserter.Drive.PLS.Up.LowLimit := 0.0;
   DropInserter.Drive.PLS.Up.HighLimit := 0.0;
   DropInserter.Drive.PLS.Up.Ok := FALSE;
   DropInserter.Drive.PLS.Intermediate.LowLimit := 0.0;
   DropInserter.Drive.PLS.Intermediate.HighLimit := 0.0;
   DropInserter.Drive.PLS.Intermediate.Ok := FALSE;
   DropInserter.Drive.PLS.Down.LowLimit := 0.0;
   DropInserter.Drive.PLS.Down.HighLimit := 0.0;
   DropInserter.Drive.PLS.Down.Ok := FALSE;
   DropInserter.Drive.PLS.Forward.LowLimit := 0.0;
   DropInserter.Drive.PLS.Forward.HighLimit := 0.0;
   DropInserter.Drive.PLS.Forward.Ok := FALSE;
   DropInserter.Drive.PLS.Backward.LowLimit := 0.0;
   DropInserter.Drive.PLS.Backward.HighLimit := 0.0;
   DropInserter.Drive.PLS.Backward.Ok := FALSE;
   DropInserter.Drive.PLS.Open.LowLimit := 0.0;
   DropInserter.Drive.PLS.Open.HighLimit := 0.0;
   DropInserter.Drive.PLS.Open.Ok := FALSE;
   DropInserter.Drive.PLS.Close.LowLimit := 0.0;
   DropInserter.Drive.PLS.Close.HighLimit := 0.0;
   DropInserter.Drive.PLS.Close.Ok := FALSE;
   DropInserter.Drive.PLS.PreOpen.LowLimit := 0.0;
   DropInserter.Drive.PLS.PreOpen.HighLimit := 0.0;
   DropInserter.Drive.PLS.PreOpen.Ok := FALSE;
   DropInserter.Drive.PLS.Maintenance.LowLimit := 0.0;
   DropInserter.Drive.PLS.Maintenance.HighLimit := 0.0;
   DropInserter.Drive.PLS.Maintenance.Ok := FALSE;
   DropInserter.Drive.PLS.OperatorSide.LowLimit := 0.0;
   DropInserter.Drive.PLS.OperatorSide.HighLimit := 0.0;
   DropInserter.Drive.PLS.OperatorSide.Ok := FALSE;
   DropInserter.Drive.PLS.NotOperatorSide.LowLimit := 0.0;
